   // ============================================================
   // 9. Перевірка положення відносно контрольних точок
   // ============================================================

   // TRUE  - координата знаходиться між контрольними точками.
   // FALSE - координата знаходиться поза ними,
   //         тому використовується лінійна екстраполяція.
   //
   // Вихід за межі контрольних точок НЕ є причиною
   // для заборони розрахунку preset.

   #InConfiguredRange :=
   (#Position_mm >= #PositionMinimum_mm)
   AND
   (#Position_mm <= #PositionMaximum_mm);

   IF NOT #InConfiguredRange THEN

       // Bit 4:
       // Цільова координата знаходиться поза діапазоном
       // двох контрольних точок.
       //
       // Це інформаційний/діагностичний біт.
       // Розрахунок продовжується методом екстраполяції.
       #Status := #Status OR W#16#0010;

   END_IF;


   // ============================================================
   // 10. Перетворення координати у raw
   // ============================================================

   #PositionDelta_mm :=
   #Position_mm
   - #PositionPoint1_mm;


   // Зворотна формула до FC_EncoderScale:
   //
   // Raw = RawPoint1
   //     + (Position - PositionPoint1)
   //       * RawSpan / PositionSpan

   #CalculatedRaw :=
   DINT_TO_LREAL(#RawPoint1)
   +
   (
   #PositionDelta_mm
   * #RawSpan
   / #PositionSpan_mm
   );

   #CalculationValid := TRUE;


   // ============================================================
   // 11. Перевірка фізично допустимого raw-діапазону
   // ============================================================

   // Саме ця перевірка є остаточним обмеженням
   // для можливості виконання hardware preset.

   #InRawRange :=
   (#CalculatedRaw >= DINT_TO_LREAL(#RawMinimum))
   AND
   (#CalculatedRaw <= DINT_TO_LREAL(#RawMaximum));

   IF NOT #InRawRange THEN

       // Bit 5:
       // Розраховане raw знаходиться поза
       // допустимим діапазоном енкодера.
       #Status := #Status OR W#16#0020;

       RETURN;

   END_IF;


   // ============================================================
   // 12. Перетворення розрахованого raw у DINT
   // ============================================================

   // Перетворення виконується тільки після перевірки
   // RawMinimum ... RawMaximum.
   //
   // Оскільки RawMinimum та RawMaximum мають тип DINT,
   // після успішної перевірки значення безпечно
   // перетворювати у DINT.

   #RawPosition :=
   LREAL_TO_DINT(#CalculatedRaw);


   // ============================================================
   // 13. Формування фінальної валідності
   // ============================================================

   // InConfiguredRange тут навмисно НЕ використовується.
   //
   // Координата може знаходитися поза двома контрольними
   // точками масштабування. У такому випадку використовується
   // лінійна екстраполяція.
   //
   // Для дозволу preset необхідно:
   // - коректна конфігурація;
   // - виконаний розрахунок;
   // - розраховане raw знаходиться у допустимих межах.

   #RawPositionValid :=
   #ConfigurationValid
   AND
   #CalculationValid
   AND
   #InRawRange;

   IF #RawPositionValid THEN

       // Bit 7:
       // Raw-значення валідне та може використовуватись
       // для hardware preset енкодера.
       #Status := #Status OR W#16#0080;

   END_IF;
END_FUNCTION

// folder: 700_Calibration/Crane

FUNCTION_BLOCK "FB_CraneCalibration"   // FB703, SCL
{ S7_Optimized_Access := 'TRUE' }
VERSION : 0.1
   VAR_INPUT
      ix_Start : Bool := FALSE;   // Запуск процедури калібровки моста
      ix_Reset : Bool := FALSE;   // Скидання сіквенсера поточної процедури калібровки (без зміни статусу)
      ix_Abort : Bool := FALSE;   // Ручне переривання процедури
      ix_ForceCalibrated : Bool := FALSE;   // Примусове встановлення статусу калібровки для ПНР
      ix_HoistCalibrated : Bool := FALSE;   // Механізм підйому відкалібрований
      ix_TrolleyCalibrated : Bool := FALSE;   // Механізм візка відкалібрований
      il_HoistPosition_mm : LReal := 0.0;   // Поточна координата механізму підйому, мм
      il_HoistPositionMin_mm : LReal := 23750.0;   // Нижня межа допустимого положення підйому для калібровки моста
      il_HoistPositionMax_mm : LReal := 23900.0;   // Верхня межа допустимого положення підйому для калібровки моста
      ix_Reference4K1 : Bool := FALSE;   // Реперний сигнал 4K1 — дозвіл номінальної швидкості при русі вліво
      ix_BtnRight : Bool := FALSE;   // Команда руху моста вправо
      ix_BtnLeft : Bool := FALSE;   // Команда руху моста вліво
      ix_Drive1Fault : Bool := FALSE;   // Аварія частотного перетворювача 4UZ1
      ix_Drive2Fault : Bool := FALSE;   // Аварія частотного перетворювача 4UZ2
      ir_Drive1Velocity_rpm : Real := 0.0;   // Фактична швидкість привода 4UZ1, об/хв
      ir_Drive2Velocity_rpm : Real := 0.0;   // Фактична швидкість привода 4UZ2, об/хв
      ix_Encoder1Ready : Bool := FALSE;   // Енкодер 4BR1 готовий
      ix_Encoder2Ready : Bool := FALSE;   // Енкодер 4BR2 готовий
      ix_Encoder1Fault : Bool := FALSE;   // Помилка енкодера 4BR1
      ix_Encoder2Fault : Bool := FALSE;   // Помилка енкодера 4BR2
      ix_Preset1Busy : Bool := FALSE;   // Виконується preset енкодера 4BR1
      ix_Preset1Done : Bool := FALSE;   // Preset енкодера 4BR1 успішно завершено
      ix_Preset1Error : Bool := FALSE;   // Помилка preset енкодера 4BR1
      iw_Preset1Status : Word := W#16#0000;   // Статус виконання preset енкодера 4BR1
      ix_Preset2Busy : Bool := FALSE;   // Виконується preset енкодера 4BR2
      ix_Preset2Done : Bool := FALSE;   // Preset енкодера 4BR2 успішно завершено
      ix_Preset2Error : Bool := FALSE;   // Помилка preset енкодера 4BR2
      iw_Preset2Status : Word := W#16#0000;   // Статус виконання preset енкодера 4BR2
      id_PresetValueRaw1 : DInt := DINT#11061828;   // Розраховане raw-значення для preset енкодера 4BR1.
      id_PresetValueRaw2 : DInt := DINT#11061828;   // Розраховане raw-значення для preset енкодера 4BR2.
      it_TimeoutA : Time := T#1m;   // Максимальний час очікування першої команди руху
      it_TimeoutB : Time := T#5m;   // Максимальний час виконання реперної процедури
      ir_StandstillSpeed_rpm : Real := 5.0;   // Максимальна швидкість привода для визначення стану standstill
      it_StandstillConfirm : Time := T#500ms;   // Час підтвердження повної зупинки обох приводів
      id_ActualPositionRaw1 : DInt := 0;   // Поточне raw-положення енкодера 4BR1
      id_ActualPositionRaw2 : DInt := 0;   // Поточне raw-положення енкодера 4BR2
      il_Scale1_mm_per_count : LReal := 0.0;   // Масштаб 4BR1, мм/count
      il_Scale2_mm_per_count : LReal := 0.0;   // Масштаб 4BR2, мм/count
      ix_PositionScale1Valid : Bool := FALSE;   // Валідність масштабування 4BR1
      ix_PositionScale2Valid : Bool := FALSE;   // Валідність масштабування 4BR2
   END_VAR
   VAR_OUTPUT
      qx_Active : Bool := FALSE;   // Процедура калібровки моста активна
      qx_Calibrated : Bool := FALSE;   // Механізм моста відкалібрований
      qx_Aborted : Bool := FALSE;   // Процедуру калібровки перервано
      qx_Fault : Bool := FALSE;   // Помилка процедури калібровки
      qx_PrerequisitesNotOK : Bool := FALSE;   // Не виконані попередні умови для калібровки моста
      qu_CurrentStep : UInt := UINT#0;   // Поточний крок сіквенсера калібровки
      qd_CompletedSteps : DWord := DWORD#0;   // Бітова маска завершених кроків калібровки
      qt_StepElapsed : Time := T#0ms;   // Час перебування на поточному кроці
      qt_ActiveTimerElapsed : Time := T#0ms;   // Поточний час активного контрольного таймера
      qt_ActiveTimerPreset : Time := T#0ms;   // Уставка активного контрольного таймера
      qt_ActiveTimerRemaining : Time := T#0ms;   // Залишок часу активного контрольного таймера
      qx_BlockRight : Bool := FALSE;   // Заборона руху моста вправо від сіквенсера калібровки
      qx_BlockLeft : Bool := FALSE;   // Заборона руху моста вліво від сіквенсера калібровки
      qx_QuickStop : Bool := FALSE;   // Запит Quick Stop для обох приводів моста
      qx_DriveStandstill : Bool := FALSE;   // Підтверджена повна зупинка обох приводів
      qx_PresetServiceEnable : Bool := FALSE;   // Загальний дозвіл preset для 4BR1 та 4BR2
      qx_PresetPermit : Bool := FALSE;   // Загальний дозвіл виконання preset для 4BR1 та 4BR2
      qx_PresetStart : Bool := FALSE;   // Загальний одноцикловий запуск preset для 4BR1 та 4BR2
      qd_PresetValueRaw1 : DInt := DINT#0;   // Значення preset, передане енкодеру 4BR1
      qd_PresetValueRaw2 : DInt := DINT#0;   // Значення preset, передане енкодеру 4BR2
      qw_Preset1Status : Word := W#16#0000;   // Поточний статус preset енкодера 4BR1
      qw_Preset2Status : Word := W#16#0000;   // Поточний статус preset енкодера 4BR2
      qw_Status : Word := W#16#0000;   // Загальне діагностичне слово стану блока калібровки
      ql_TravelAfterReference1_mm : LReal := 0.0;   // Шлях, пройдений після повторного проходження 4K1 до повної зупинки (4BR1), мм.
      ql_TravelAfterReference2_mm : LReal := 0.0;   // Шлях, пройдений після повторного проходження 4K1 до повної зупинки (4BR2), мм.
   END_VAR
   VAR
      stat_Step : UInt := UINT#0;   // Поточний внутрішній крок сіквенсера
      stat_PrevStep : UInt := UINT#0;   // Попередній крок для визначення зміни кроку
   END_VAR
   VAR RETAIN
      stat_Calibrated : Bool := FALSE;   // Запам'ятований результат успішної калібровки моста
   END_VAR
   VAR
      stat_MotionStarted : Bool := FALSE;   // Ознака, що під час процедури вже була команда руху
      stat_CompletedSteps : DWord := DWORD#0;   // Внутрішня бітова маска завершених кроків
      stat_StartOld : Bool := FALSE;   // Попередній стан команди Start
      stat_ResetOld : Bool := FALSE;   // Попередній стан команди Reset
      stat_AbortOld : Bool := FALSE;   // Попередній стан команди Abort
      stat_ReferenceOld : Bool := FALSE;   // Попередній стан реперного сигналу 4K1
      tmr_TimeoutA : TON_TIME;   // Таймер очікування першої команди руху
      tmr_TimeoutB : TON_TIME;   // Таймер максимальної тривалості реперної процедури
      tmr_Standstill : TON_TIME;   // Таймер підтвердження повної зупинки обох ПЧ
      tmr_StepElapsed : TON_TIME;   // Таймер часу перебування на поточному кроці
      stat_RawAtReference1 : DInt := 0;   // Raw-положення енкодера 4BR1 в момент повторного спадного фронту 4K1.
      stat_RawAtReference2 : DInt := 0;   // Raw-положення енкодера 4BR2 в момент повторного спадного фронту 4K1.
      stat_RawAtReference1Valid : Bool := FALSE;   // TRUE - raw-положення 4BR1 в точці 4K1 успішно зафіксовано.
      stat_RawAtReference2Valid : Bool := FALSE;   // TRUE - raw-положення 4BR2 в точці 4K1 успішно зафіксовано.
      stat_TravelAfterReference1_mm : LReal := 0.0;   // Розрахований шлях 4BR1 від 4K1 до повної зупинки.
      stat_TravelAfterReference2_mm : LReal := 0.0;   // Розрахований шлях 4BR2 від 4K1 до повної зупинки.
   END_VAR
   VAR_TEMP
      StartEdge : Bool;   // Передній фронт команди запуску калібровки
      ResetEdge : Bool;   // Передній фронт команди Reset
      AbortEdge : Bool;   // Передній фронт команди Abort
      ReferenceFalling : Bool;   // Спадний фронт 4K1, тобто проходження реперної точки при русі вліво
      StepChanged : Bool;   // Ознака зміни поточного кроку сіквенсера
      StandstillCondition : Bool;   // Обидва приводи мають швидкість нижче порога standstill
      HoistPositionOK : Bool;   // Підйом калібрований та знаходиться в допустимій зоні
      PrerequisitesOK : Bool;   // Виконані всі попередні умови для калібровки моста
   END_VAR
BEGIN
   // ============================================================
   // 1. Формування фронтів
   // ============================================================

   #StartEdge :=
   #ix_Start
   AND NOT #stat_StartOld;

   #ResetEdge :=
   #ix_Reset
   AND NOT #stat_ResetOld;

   #AbortEdge :=
   #ix_Abort
   AND NOT #stat_AbortOld;

   // 4K1: проходження репера при русі вліво.
   // Сигнал змінюється TRUE -> FALSE.
   #ReferenceFalling :=
   #stat_ReferenceOld
   AND NOT #ix_Reference4K1;


   // ============================================================
   // 2. Початкові умови калібровки моста
   // ============================================================

   #HoistPositionOK :=
   #ix_HoistCalibrated
   AND (#il_HoistPosition_mm >= #il_HoistPositionMin_mm)
   AND (#il_HoistPosition_mm <= #il_HoistPositionMax_mm);

   #PrerequisitesOK :=
   #HoistPositionOK
   AND #ix_TrolleyCalibrated;

   #qx_PrerequisitesNotOK :=
   NOT #PrerequisitesOK;


   // ============================================================
   // 3. Reset
   // ============================================================

   IF #ResetEdge THEN

       #stat_Step := UINT#0;
       #stat_PrevStep := UINT#0;

       #stat_MotionStarted := FALSE;
       #stat_CompletedSteps := DWORD#0;

       #stat_RawAtReference1 := DINT#0;
       #stat_RawAtReference2 := DINT#0;

       #stat_RawAtReference1Valid := FALSE;
       #stat_RawAtReference2Valid := FALSE;

       #stat_TravelAfterReference1_mm := 0.0;
       #stat_TravelAfterReference2_mm := 0.0;


   END_IF;


   // ============================================================
   // 4. Timeout A
   // ============================================================

   #tmr_TimeoutA(
                 IN :=
                 (#stat_Step = UINT#5)
                 OR (#stat_Step = UINT#20)
                 OR (#stat_Step = UINT#50)
                 OR (#stat_Step = UINT#70),
                 PT := #it_TimeoutA
   );


   // ============================================================
   // 5. Timeout B
   // ============================================================

   #tmr_TimeoutB(
                 IN :=
                 (#stat_Step = UINT#30)
                 OR (#stat_Step = UINT#80),
                 PT := #it_TimeoutB
   );


   // ============================================================
   // 6. Контроль повної зупинки обох приводів
   // ============================================================

   #StandstillCondition :=
   (ABS(#ir_Drive1Velocity_rpm) <= #ir_StandstillSpeed_rpm)
   AND
   (ABS(#ir_Drive2Velocity_rpm) <= #ir_StandstillSpeed_rpm);

   #tmr_Standstill(
                   IN :=
                   (#stat_Step >= UINT#100)
                   AND (#stat_Step <= UINT#120)
                   AND #StandstillCondition,
                   PT := #it_StandstillConfirm
   );

   #qx_DriveStandstill :=
   #tmr_Standstill.Q;


   // ============================================================
   // 7. Таймер поточного кроку
   // ============================================================

   #StepChanged :=
   #stat_Step <> #stat_PrevStep;

   #tmr_StepElapsed(
                    IN :=
                    (#stat_Step > UINT#0)
                    AND (#stat_Step < UINT#130)
                    AND NOT #StepChanged,
                    PT := T#24d
   );

   #qt_StepElapsed :=
   #tmr_StepElapsed.ET;

   IF #StepChanged THEN
       #stat_PrevStep := #stat_Step;
   END_IF;


   // ============================================================
   // 8. Виходи за замовчуванням
   // ============================================================

   #qx_Active := FALSE;
   #qx_Aborted := FALSE;
   #qx_Fault := FALSE;

   #qx_BlockRight := TRUE;
   #qx_BlockLeft := TRUE;

   #qx_QuickStop := FALSE;

   #qx_PresetServiceEnable := FALSE;
   #qx_PresetPermit := FALSE;
   #qx_PresetStart := FALSE;

   #qd_PresetValueRaw1 :=
   #id_PresetValueRaw1;

   #qd_PresetValueRaw2 :=
   #id_PresetValueRaw2;

   #qw_Preset1Status :=
   #iw_Preset1Status;

   #qw_Preset2Status :=
   #iw_Preset2Status;


   // ============================================================
   // 9. Загальні умови аварійного завершення
   //
   // Працюють тільки під час активної процедури.
   // STEP 130 після успішної калібровки не переводиться в 910.
   // ============================================================

   IF (#stat_Step > UINT#0)
       AND (#stat_Step < UINT#130)
   THEN

       IF #AbortEdge THEN

           #stat_Step := UINT#900;

       ELSIF #ix_Drive1Fault
           OR #ix_Drive2Fault
           OR #ix_Encoder1Fault
           OR #ix_Encoder2Fault
       THEN

           #stat_Step := UINT#910;

           // Підйом і візок повинні залишатися
           // у допустимому стані під час процедури.
       ELSIF NOT #PrerequisitesOK THEN

           #stat_Step := UINT#910;

       ELSIF (#stat_Step < UINT#110)
           AND (
           NOT #ix_Encoder1Ready
           OR NOT #ix_Encoder2Ready
           )
       THEN

           #stat_Step := UINT#910;

       ELSIF #tmr_TimeoutA.Q THEN

           #stat_Step := UINT#910;

       ELSIF #tmr_TimeoutB.Q THEN

           #stat_Step := UINT#910;

       END_IF;

   END_IF;


   // ============================================================
   // 10. Основний сіквенсер
   // ============================================================

   CASE #stat_Step OF


           // --------------------------------------------------------
           // STEP 0
           // Калібровка неактивна
           // --------------------------------------------------------
       UINT#0:

           #qx_BlockRight := FALSE;
           #qx_BlockLeft := FALSE;

           IF #StartEdge THEN

               #stat_Calibrated := FALSE;
               #stat_MotionStarted := FALSE;
               #stat_CompletedSteps := DWORD#0;

               #stat_RawAtReference1 := DINT#0;
               #stat_RawAtReference2 := DINT#0;

               #stat_RawAtReference1Valid := FALSE;
               #stat_RawAtReference2Valid := FALSE;

               #stat_TravelAfterReference1_mm := 0.0;
               #stat_TravelAfterReference2_mm := 0.0;

               IF #PrerequisitesOK THEN

                   // Нормальний старт перед репером 4K1.
                   IF #ix_Reference4K1 THEN

                       #stat_Step := UINT#10;

                       // Якщо механізм вже знаходиться на / за 4K1,
                       // спочатку необхідно відійти вправо.
                   ELSE

                       #stat_Step := UINT#5;

                   END_IF;

               ELSE

                   #stat_Step := UINT#910;

               END_IF;

           END_IF;


           // --------------------------------------------------------
           // STEP 5
           // Попередній відхід вправо від 4K1
           // --------------------------------------------------------
       UINT#5:

           #qx_Active := TRUE;

           // До репера вліво рух заборонений.
           // Дозволений тільки відхід вправо.
           #qx_BlockRight := FALSE;
           #qx_BlockLeft := TRUE;

           IF #ix_BtnRight THEN
               #stat_MotionStarted := TRUE;
           END_IF;

           // Після звільнення 4K1 та відпускання кнопки
           // запускаємо штатну процедуру.
           IF #ix_Reference4K1
               AND NOT #ix_BtnRight
           THEN

               #stat_Step := UINT#10;

           END_IF;


           // --------------------------------------------------------
           // STEP 10
           // Перевірка початкових умов
           // --------------------------------------------------------
       UINT#10:

           #qx_Active := TRUE;

           #qx_BlockRight := TRUE;
           #qx_BlockLeft := TRUE;

           IF NOT #ix_BtnRight
               AND NOT #ix_BtnLeft
           THEN

               #stat_CompletedSteps.%X0 := TRUE;
               #stat_Step := UINT#20;

           END_IF;


           // --------------------------------------------------------
           // STEP 20
           // Очікування першої команди "Вліво"
           // --------------------------------------------------------
       UINT#20:

           #qx_Active := TRUE;

           #qx_BlockRight := TRUE;
           #qx_BlockLeft := FALSE;

           IF #ix_BtnLeft THEN

               #stat_MotionStarted := TRUE;
               #stat_CompletedSteps.%X1 := TRUE;

               #stat_Step := UINT#30;

           END_IF;


           // --------------------------------------------------------
           // STEP 30
           // Перший рух вліво до 4K1
           // --------------------------------------------------------
       UINT#30:

           #qx_Active := TRUE;

           #qx_BlockRight := TRUE;
           #qx_BlockLeft := FALSE;

           IF #ReferenceFalling THEN

               #stat_CompletedSteps.%X2 := TRUE;
               #stat_Step := UINT#40;

           END_IF;


           // --------------------------------------------------------
           // STEP 40
           // Перше проходження 4K1
           // Очікування відпускання кнопки "Вліво"
           // --------------------------------------------------------
       UINT#40:

           #qx_Active := TRUE;

           #qx_BlockRight := TRUE;
           #qx_BlockLeft := TRUE;

           IF NOT #ix_BtnLeft THEN

               #stat_CompletedSteps.%X3 := TRUE;
               #stat_Step := UINT#50;

           END_IF;


           // --------------------------------------------------------
           // STEP 50
           // Відхід вправо від репера
           // --------------------------------------------------------
       UINT#50:

           #qx_Active := TRUE;

           #qx_BlockRight := FALSE;
           #qx_BlockLeft := TRUE;

           IF #ix_BtnRight THEN
               #stat_MotionStarted := TRUE;
           END_IF;

           IF #ix_Reference4K1
               AND NOT #ix_BtnRight
           THEN

               #stat_CompletedSteps.%X4 := TRUE;
               #stat_Step := UINT#60;

           END_IF;


           // --------------------------------------------------------
           // STEP 60
           // Репер звільнений
           // --------------------------------------------------------
       UINT#60:

           #qx_Active := TRUE;

           #qx_BlockRight := TRUE;
           #qx_BlockLeft := TRUE;

           #stat_CompletedSteps.%X5 := TRUE;
           #stat_Step := UINT#70;


           // --------------------------------------------------------
           // STEP 70
           // Очікування повторної команди "Вліво"
           // --------------------------------------------------------
       UINT#70:

           #qx_Active := TRUE;

           #qx_BlockRight := TRUE;
           #qx_BlockLeft := FALSE;

           IF #ix_BtnLeft THEN

               #stat_CompletedSteps.%X6 := TRUE;
               #stat_Step := UINT#80;

           END_IF;


           // --------------------------------------------------------
           // STEP 80
           // Повторний точний підхід вліво до 4K1
           // --------------------------------------------------------
       UINT#80:

           #qx_Active := TRUE;

           #qx_BlockRight := TRUE;
           #qx_BlockLeft := FALSE;

           IF #ReferenceFalling THEN

               // Обидва канали масштабування повинні бути валідні.
               IF #ix_PositionScale1Valid
                   AND #ix_PositionScale2Valid
               THEN

                   // Одночасно запам'ятовуємо raw-положення
                   // обох енкодерів у момент проходження 4K1.
                   #stat_RawAtReference1 :=
                   #id_ActualPositionRaw1;

                   #stat_RawAtReference2 :=
                   #id_ActualPositionRaw2;

                   #stat_RawAtReference1Valid := TRUE;
                   #stat_RawAtReference2Valid := TRUE;

                   #stat_CompletedSteps.%X7 := TRUE;
                   #stat_Step := UINT#90;

               ELSE

                   #stat_RawAtReference1Valid := FALSE;
                   #stat_RawAtReference2Valid := FALSE;

                   #stat_Step := UINT#910;

               END_IF;

           END_IF;



           // --------------------------------------------------------
           // STEP 90
           // Quick Stop обох приводів
           // --------------------------------------------------------
       UINT#90:

           #qx_Active := TRUE;

           #qx_BlockRight := TRUE;
           #qx_BlockLeft := TRUE;
           #qx_QuickStop := TRUE;

           #stat_CompletedSteps.%X8 := TRUE;

           #stat_Step := UINT#100;


           // --------------------------------------------------------
           // STEP 100
           // Очікування повної зупинки обох приводів
           // --------------------------------------------------------
       UINT#100:

           #qx_Active := TRUE;

           #qx_BlockRight := TRUE;
           #qx_BlockLeft := TRUE;

           #qx_QuickStop := TRUE;

           IF #qx_DriveStandstill
               AND NOT #ix_BtnRight
               AND NOT #ix_BtnLeft
           THEN

               IF #stat_RawAtReference1Valid
                   AND #stat_RawAtReference2Valid
                   AND #ix_PositionScale1Valid
                   AND #ix_PositionScale2Valid
               THEN

                   // Шлях 4BR1 від проходження 4K1
                   // до підтвердженої повної зупинки.
                   #stat_TravelAfterReference1_mm :=
                   (
                   DINT_TO_LREAL(#id_ActualPositionRaw1)
                   - DINT_TO_LREAL(#stat_RawAtReference1)
                   )
                   * #il_Scale1_mm_per_count;

                   // Шлях 4BR2 від проходження 4K1
                   // до підтвердженої повної зупинки.
                   #stat_TravelAfterReference2_mm :=
                   (
                   DINT_TO_LREAL(#id_ActualPositionRaw2)
                   - DINT_TO_LREAL(#stat_RawAtReference2)
                   )
                   * #il_Scale2_mm_per_count;

                   #stat_CompletedSteps.%X9 := TRUE;
                   #stat_Step := UINT#110;

               ELSE

                   #stat_Step := UINT#910;

               END_IF;

           END_IF;


           // --------------------------------------------------------
           // STEP 110
           // Запуск preset обох енкодерів
           // --------------------------------------------------------
       UINT#110:

           #qx_Active := TRUE;

           #qx_BlockRight := TRUE;
           #qx_BlockLeft := TRUE;

           #qx_PresetServiceEnable := TRUE;

           #qx_PresetPermit :=
           #qx_DriveStandstill
           AND NOT #ix_BtnRight
           AND NOT #ix_BtnLeft
           AND #ix_Encoder1Ready
           AND #ix_Encoder2Ready
           AND NOT #ix_Encoder1Fault
           AND NOT #ix_Encoder2Fault
           AND NOT #ix_Drive1Fault
           AND NOT #ix_Drive2Fault;

           IF #qx_PresetPermit THEN

               // Один імпульс одночасно запускає preset
               // для 4BR1 та 4BR2.
               #qx_PresetStart := TRUE;

               #stat_CompletedSteps.%X10 := TRUE;
               #stat_Step := UINT#120;

           END_IF;


           // --------------------------------------------------------
           // STEP 120
           // Очікування завершення preset обох енкодерів
           // --------------------------------------------------------
       UINT#120:

           #qx_Active := TRUE;

           #qx_BlockRight := TRUE;
           #qx_BlockLeft := TRUE;

           #qx_PresetServiceEnable := TRUE;

           #qx_PresetPermit :=
           #qx_DriveStandstill
           AND NOT #ix_BtnRight
           AND NOT #ix_BtnLeft
           AND NOT #ix_Encoder1Fault
           AND NOT #ix_Encoder2Fault
           AND NOT #ix_Drive1Fault
           AND NOT #ix_Drive2Fault;

           // Обидва preset повинні завершитися успішно.
           IF #ix_Preset1Done
               AND #ix_Preset2Done
           THEN

               #stat_CompletedSteps.%X11 := TRUE;
               #stat_Step := UINT#130;

           ELSIF #ix_Preset1Error
               OR #ix_Preset2Error
           THEN

               #stat_Step := UINT#910;

           END_IF;


           // --------------------------------------------------------
           // STEP 130
           // Калібровка моста успішно завершена
           // --------------------------------------------------------
       UINT#130:

           #qx_BlockRight := FALSE;
           #qx_BlockLeft := FALSE;

           #stat_Calibrated := TRUE;
           #stat_CompletedSteps.%X12 := TRUE;


           // --------------------------------------------------------
           // STEP 900
           // Ручне переривання
           // --------------------------------------------------------
       UINT#900:

           #qx_Aborted := TRUE;

           #qx_BlockRight := TRUE;
           #qx_BlockLeft := TRUE;

           #qx_QuickStop := TRUE;


           // --------------------------------------------------------
           // STEP 910
           // Помилка процедури
           // --------------------------------------------------------
       UINT#910:

           #qx_Fault := TRUE;

           #qx_BlockRight := TRUE;
           #qx_BlockLeft := TRUE;

           #qx_QuickStop := TRUE;


       ELSE

           #stat_Step := UINT#910;

   END_CASE;


   // ============================================================
   // 11. Основні статуси
   // ============================================================

   #qu_CurrentStep :=
   #stat_Step;

   #qd_CompletedSteps :=
   #stat_CompletedSteps;

   #qx_Calibrated :=
   #stat_Calibrated
   OR #ix_ForceCalibrated;

   #ql_TravelAfterReference1_mm :=
   #stat_TravelAfterReference1_mm;

   #ql_TravelAfterReference2_mm :=
   #stat_TravelAfterReference2_mm;

   // ============================================================
   // 12. Активний таймер для HMI
   // ============================================================

   #qt_ActiveTimerElapsed := T#0ms;
   #qt_ActiveTimerPreset := T#0ms;
   #qt_ActiveTimerRemaining := T#0ms;

   // Timeout A
   IF (#stat_Step = UINT#5)
       OR (#stat_Step = UINT#20)
       OR (#stat_Step = UINT#50)
       OR (#stat_Step = UINT#70)
   THEN

       #qt_ActiveTimerElapsed :=
       #tmr_TimeoutA.ET;

       #qt_ActiveTimerPreset :=
       #it_TimeoutA;

       IF #tmr_TimeoutA.ET < #it_TimeoutA THEN

           #qt_ActiveTimerRemaining :=
           #it_TimeoutA - #tmr_TimeoutA.ET;

       END_IF;


       // Timeout B
   ELSIF 
       (#stat_Step = UINT#30)
       OR (#stat_Step = UINT#80)
   THEN

       #qt_ActiveTimerElapsed :=
       #tmr_TimeoutB.ET;

       #qt_ActiveTimerPreset :=
       #it_TimeoutB;

       IF #tmr_TimeoutB.ET < #it_TimeoutB THEN

           #qt_ActiveTimerRemaining :=
           #it_TimeoutB - #tmr_TimeoutB.ET;

       END_IF;


       // Standstill
   ELSIF #stat_Step = UINT#100 THEN

       #qt_ActiveTimerElapsed :=
       #tmr_Standstill.ET;

       #qt_ActiveTimerPreset :=
       #it_StandstillConfirm;

       IF #tmr_Standstill.ET < #it_StandstillConfirm THEN

           #qt_ActiveTimerRemaining :=
           #it_StandstillConfirm - #tmr_Standstill.ET;

       END_IF;

   END_IF;


   // ============================================================
   // 13. Діагностичне слово
   // ============================================================

   #qw_Status := W#16#0000;

   IF #qx_Active THEN
       #qw_Status := #qw_Status OR W#16#0001;
   END_IF;

   IF #qx_Calibrated THEN
       #qw_Status := #qw_Status OR W#16#0002;
   END_IF;

   IF #qx_Aborted THEN
       #qw_Status := #qw_Status OR W#16#0004;
   END_IF;

   IF #qx_Fault THEN
       #qw_Status := #qw_Status OR W#16#0008;
   END_IF;

   IF #qx_DriveStandstill THEN
       #qw_Status := #qw_Status OR W#16#0010;
   END_IF;

   IF #ix_Preset1Busy OR #ix_Preset2Busy THEN
       #qw_Status := #qw_Status OR W#16#0020;
   END_IF;

   IF #ix_Preset1Error OR #ix_Preset2Error THEN
       #qw_Status := #qw_Status OR W#16#0040;
   END_IF;

   IF #qx_PrerequisitesNotOK THEN
       #qw_Status := #qw_Status OR W#16#0080;
   END_IF;

   IF #tmr_TimeoutA.Q THEN
       #qw_Status := #qw_Status OR W#16#0100;
   END_IF;

   IF #tmr_TimeoutB.Q THEN
       #qw_Status := #qw_Status OR W#16#0200;
   END_IF;

   IF #ix_Drive1Fault OR #ix_Drive2Fault THEN
       #qw_Status := #qw_Status OR W#16#0400;
   END_IF;

   IF #ix_Encoder1Fault OR #ix_Encoder2Fault THEN
       #qw_Status := #qw_Status OR W#16#0800;
   END_IF;

   IF NOT #ix_Encoder1Ready
       OR NOT #ix_Encoder2Ready
   THEN
       #qw_Status := #qw_Status OR W#16#1000;
   END_IF;


   // ============================================================
   // 14. Запам'ятовування станів
   // ============================================================

   #stat_StartOld :=
   #ix_Start;

   #stat_ResetOld :=
   #ix_Reset;

   #stat_AbortOld :=
   #ix_Abort;

   #stat_ReferenceOld :=
   #ix_Reference4K1;
END_FUNCTION_BLOCK

FUNCTION_BLOCK "FB_CraneCalibrationDiag"   // FB713, SCL
{ S7_Optimized_Access := 'TRUE' }
VERSION : 0.1
   VAR_INPUT
      ix_Reset : Bool := FALSE;   // Скидання зафіксованих діагностичних помилок
      ix_Encoder1Ready : Bool := FALSE;   // Енкодер 4BR1 готовий
      ix_Encoder1Fault : Bool := FALSE;   // Помилка енкодера 4BR1
      ix_Communication1Fault : Bool := FALSE;   // Помилка зв'язку з енкодером 4BR1
      il_Position1_mm : LReal := 0.0;   // Поточна координата за енкодером 4BR1, мм
      ix_Encoder2Ready : Bool := FALSE;   // Енкодер 4BR2 готовий
      ix_Encoder2Fault : Bool := FALSE;   // Помилка енкодера 4BR2
      ix_Communication2Fault : Bool := FALSE;   // Помилка зв'язку з енкодером 4BR2
      il_Position2_mm : LReal := 0.0;   // Поточна координата за енкодером 4BR2, мм
      ix_MoveCommand : Bool := FALSE;   // Дійсна команда руху моста
      ix_Drive1Fault : Bool := FALSE;   // Аварія привода 4UZ1
      ix_Drive2Fault : Bool := FALSE;   // Аварія привода 4UZ2
      ir_Drive1Velocity_rpm : Real := 0.0;   // Фактична швидкість 4UZ1, об/хв
      ir_Drive2Velocity_rpm : Real := 0.0;   // Фактична швидкість 4UZ2, об/хв
      ix_CalibrationActive : Bool := FALSE;   // Процедура калібровки моста активна
      ix_Calibrated : Bool := FALSE;   // Міст відкалібрований
      ix_ManualDriveActive : Bool := FALSE;   // Ручний привод активний; поки FALSE
      il_NoMoveThreshold_mm : LReal := 5.0;   // Допустима зміна положення без команди
      il_MoveMinDelta_mm : LReal := 1.0;   // Мінімальна зміна координати при русі
      it_MoveUpdateTimeout : Time := T#1s;   // Максимальний час без зміни координати
      ir_StandstillSpeed_rpm : Real := 5.0;   // Поріг повної зупинки приводів
      it_StandstillConfirm : Time := T#500ms;   // Час підтвердження повної зупинки
      il_StartupTolerance_mm : LReal := 5.0;   // Допуск перевірки координати після запуску PLC
      il_MaxEncoderDifference_mm : LReal := 50.0;   // Максимальна допустима розбіжність 4BR1 та 4BR2
   END_VAR
   VAR_OUTPUT
      qx_Encoder1ControlHealthy : Bool := FALSE;   // Енкодер 4BR1 і його зв'язок справні
      qx_Encoder1StartupDataConsistent : Bool := TRUE;   // Дані 4BR1 після старту PLC узгоджені
      qx_Encoder1NoMovementWithoutCommand : Bool := TRUE;   // Для 4BR1 не виявлено руху без команди
      qx_Encoder1NoManualMovementDetected : Bool := TRUE;   // Для 4BR1 не виявлено нештатного переміщення
      qx_Encoder1UpdatesDuringMotion : Bool := TRUE;   // 4BR1 змінює координату під час руху
      qx_Encoder1ReplacementNotDetected : Bool := TRUE;   // Заміна 4BR1 не виявлена; поки завжди норма
      qx_Encoder2ControlHealthy : Bool := FALSE;   // Енкодер 4BR2 і його зв'язок справні
      qx_Encoder2StartupDataConsistent : Bool := TRUE;   // Дані 4BR2 після старту PLC узгоджені
      qx_Encoder2NoMovementWithoutCommand : Bool := TRUE;   // Для 4BR2 не виявлено руху без команди
      qx_Encoder2NoManualMovementDetected : Bool := TRUE;   // Для 4BR2 не виявлено нештатного переміщення
      qx_Encoder2UpdatesDuringMotion : Bool := TRUE;   // 4BR2 змінює координату під час руху
      qx_Encoder2ReplacementNotDetected : Bool := TRUE;   // Заміна 4BR2 не виявлена; поки завжди норма
      qx_EncoderDifferenceOK : Bool := TRUE;   // Розбіжність координат 4BR1/4BR2 у нормі
      qx_DiagnosticsHealthy : Bool := FALSE;   // Загальний результат діагностики моста
      qx_DriveStandstill : Bool := FALSE;   // Підтверджена повна зупинка обох приводів
      ql_EncoderDifference_mm : LReal := 0.0;   // Поточна абсолютна розбіжність 4BR1/4BR2, мм
      ql_Position1DeltaStopped_mm : LReal := 0.0;   // Зміна 4BR1 від точки зупинки
      ql_Position2DeltaStopped_mm : LReal := 0.0;   // Зміна 4BR2 від точки зупинки
      ql_Position1DeltaMotion_mm : LReal := 0.0;   // Зміна 4BR1 для watchdog руху
      ql_Position2DeltaMotion_mm : LReal := 0.0;   // Зміна 4BR2 для watchdog руху
   END_VAR
   VAR RETAIN
      stat_SavedPosition1_mm : LReal := 0.0;   // Збережена до перезапуску позиція 4BR1
      stat_SavedPosition1Valid : Bool := FALSE;   // Збережена позиція 4BR1 валідна
      stat_SavedPosition2_mm : LReal := 0.0;   // Збережена до перезапуску позиція 4BR2
      stat_SavedPosition2Valid : Bool := FALSE;   // Збережена позиція 4BR2 валідна
   END_VAR
   VAR
      stat_StartupChecked : Bool := FALSE;   // Стартова перевірка виконана
      stat_StopReference1_mm : LReal := 0.0;   // Базова позиція 4BR1 після зупинки
      stat_StopReference1Valid : Bool := FALSE;   // Базова позиція 4BR1 валідна
      stat_StopReference2_mm : LReal := 0.0;   // Базова позиція 4BR2 після зупинки
      stat_StopReference2Valid : Bool := FALSE;   // Базова позиція 4BR2 валідна
      stat_MoveReference1_mm : LReal := 0.0;   // База watchdog 4BR1
      stat_MoveReference2_mm : LReal := 0.0;   // База watchdog 4BR2
      stat_MoveMonitor1Active : Bool := FALSE;   // Watchdog 4BR1 активний
      stat_MoveMonitor2Active : Bool := FALSE;   // Watchdog 4BR2 активний
      stat_WasMoving : Bool := FALSE;   // Міст до цього рухався
      stat_StartupMismatch1Fault : Bool := FALSE;   // Стартова невідповідність 4BR1
      stat_StartupMismatch2Fault : Bool := FALSE;   // Стартова невідповідність 4BR2
      stat_MoveWithoutCommand1Fault : Bool := FALSE;   // Зміна 4BR1 без команди
      stat_MoveWithoutCommand2Fault : Bool := FALSE;   // Зміна 4BR2 без команди
      stat_NoUpdateDuringMotion1Fault : Bool := FALSE;   // 4BR1 не оновлюється при русі
      stat_NoUpdateDuringMotion2Fault : Bool := FALSE;   // 4BR2 не оновлюється при русі
      stat_EncoderDifferenceFault : Bool := FALSE;   // Розбіжність енкодерів перевищила допустиму
      stat_CalibratedOld : Bool := FALSE;   // Попередній стан Calibrated
      tmr_Standstill : TON_TIME;   // Підтвердження повної зупинки
      tmr_MoveUpdate1 : TON_TIME;   // Watchdog 4BR1
      tmr_MoveUpdate2 : TON_TIME;   // Watchdog 4BR2
   END_VAR
   VAR_TEMP
      Encoder1Healthy : Bool;   // Поточна справність 4BR1
      Encoder2Healthy : Bool;   // Поточна справність 4BR2
      StandstillCondition : Bool;   // Обидва ПЧ мають низьку швидкість
      CalibratedRising : Bool;   // Передній фронт Calibrated
      MoveDelta1Reached : Bool;   // 4BR1 змінився на задану величину
      MoveDelta2Reached : Bool;   // 4BR2 змінився на задану величину
      MoveWatchdog1Enable : Bool;   // Дозвіл watchdog 4BR1
      MoveWatchdog2Enable : Bool;   // Дозвіл watchdog 4BR2
   END_VAR
BEGIN
   // ============================================================
   // 1. Справність енкодерів
   // ============================================================

   #Encoder1Healthy :=
   #ix_Encoder1Ready
   AND NOT #ix_Encoder1Fault
   AND NOT #ix_Communication1Fault;

   #Encoder2Healthy :=
   #ix_Encoder2Ready
   AND NOT #ix_Encoder2Fault
   AND NOT #ix_Communication2Fault;

   #qx_Encoder1ControlHealthy :=
   #Encoder1Healthy;

   #qx_Encoder2ControlHealthy :=
   #Encoder2Healthy;


   // ============================================================
   // 2. Визначення повної зупинки обох приводів
   // ============================================================

   #StandstillCondition :=
   (ABS(#ir_Drive1Velocity_rpm) <= #ir_StandstillSpeed_rpm)
   AND
   (ABS(#ir_Drive2Velocity_rpm) <= #ir_StandstillSpeed_rpm);

   #tmr_Standstill(
                   IN :=
                   #StandstillCondition
                   AND NOT #ix_MoveCommand,
                   PT := #it_StandstillConfirm
   );

   #qx_DriveStandstill :=
   #tmr_Standstill.Q;


   // ============================================================
   // 3. Фронт статусу "Калібровано"
   // ============================================================

   #CalibratedRising :=
   #ix_Calibrated
   AND NOT #stat_CalibratedOld;


   // ============================================================
   // 4. Reset діагностики
   // ============================================================

   IF #ix_Reset THEN

       #stat_StartupMismatch1Fault := FALSE;
       #stat_StartupMismatch2Fault := FALSE;

       #stat_MoveWithoutCommand1Fault := FALSE;
       #stat_MoveWithoutCommand2Fault := FALSE;

       #stat_NoUpdateDuringMotion1Fault := FALSE;
       #stat_NoUpdateDuringMotion2Fault := FALSE;

       #stat_EncoderDifferenceFault := FALSE;

       #stat_StopReference1Valid := FALSE;
       #stat_StopReference2Valid := FALSE;

       #stat_MoveMonitor1Active := FALSE;
       #stat_MoveMonitor2Active := FALSE;

   END_IF;


   // ============================================================
   // 5. Перевірка позицій після запуску PLC
   // ============================================================

   IF NOT #stat_StartupChecked
       AND #Encoder1Healthy
       AND #Encoder2Healthy
   THEN

       // 4BR1
       IF #stat_SavedPosition1Valid THEN

           IF ABS(#il_Position1_mm - #stat_SavedPosition1_mm)
               > #il_StartupTolerance_mm
           THEN
               #stat_StartupMismatch1Fault := TRUE;
           END_IF;

       ELSE

           #stat_SavedPosition1_mm :=
           #il_Position1_mm;

           #stat_SavedPosition1Valid := TRUE;

       END_IF;


       // 4BR2
       IF #stat_SavedPosition2Valid THEN

           IF ABS(#il_Position2_mm - #stat_SavedPosition2_mm)
               > #il_StartupTolerance_mm
           THEN
               #stat_StartupMismatch2Fault := TRUE;
           END_IF;

       ELSE

           #stat_SavedPosition2_mm :=
           #il_Position2_mm;

           #stat_SavedPosition2Valid := TRUE;

       END_IF;


       #stat_StartupChecked := TRUE;

       #stat_StopReference1_mm :=
       #il_Position1_mm;

       #stat_StopReference1Valid := TRUE;

       #stat_StopReference2_mm :=
       #il_Position2_mm;

       #stat_StopReference2Valid := TRUE;

   END_IF;


   // ============================================================
   // 6. Після успішної калібровки
   // ============================================================

   IF #CalibratedRising
       AND #Encoder1Healthy
       AND #Encoder2Healthy
   THEN

       #stat_StopReference1_mm :=
       #il_Position1_mm;

       #stat_StopReference1Valid := TRUE;

       #stat_StopReference2_mm :=
       #il_Position2_mm;

       #stat_StopReference2Valid := TRUE;


       #stat_SavedPosition1_mm :=
       #il_Position1_mm;

       #stat_SavedPosition1Valid := TRUE;

       #stat_SavedPosition2_mm :=
       #il_Position2_mm;

       #stat_SavedPosition2Valid := TRUE;


       #stat_StartupMismatch1Fault := FALSE;
       #stat_StartupMismatch2Fault := FALSE;

       #stat_MoveWithoutCommand1Fault := FALSE;
       #stat_MoveWithoutCommand2Fault := FALSE;

       #stat_NoUpdateDuringMotion1Fault := FALSE;
       #stat_NoUpdateDuringMotion2Fault := FALSE;

       #stat_EncoderDifferenceFault := FALSE;

   END_IF;


   // ============================================================
   // 7. Запам'ятовування факту руху
   // ============================================================

   IF #ix_MoveCommand THEN
       #stat_WasMoving := TRUE;
   END_IF;


   // ============================================================
   // 8. Формування нових баз після завершення руху
   // ============================================================

   IF #qx_DriveStandstill
       AND #stat_WasMoving
       AND #Encoder1Healthy
       AND #Encoder2Healthy
       AND NOT #ix_CalibrationActive
   THEN

       #stat_StopReference1_mm :=
       #il_Position1_mm;

       #stat_StopReference1Valid := TRUE;

       #stat_StopReference2_mm :=
       #il_Position2_mm;

       #stat_StopReference2Valid := TRUE;


       #stat_SavedPosition1_mm :=
       #il_Position1_mm;

       #stat_SavedPosition1Valid := TRUE;

       #stat_SavedPosition2_mm :=
       #il_Position2_mm;

       #stat_SavedPosition2Valid := TRUE;

       #stat_WasMoving := FALSE;

   END_IF;


   // ============================================================
   // 9. Контроль зміни положення без команди
   // ============================================================

   #ql_Position1DeltaStopped_mm := 0.0;
   #ql_Position2DeltaStopped_mm := 0.0;

   IF #qx_DriveStandstill
       AND NOT #ix_MoveCommand
       AND NOT #ix_ManualDriveActive
       AND NOT #ix_CalibrationActive
   THEN

       // 4BR1
       IF #Encoder1Healthy
           AND #stat_StopReference1Valid
       THEN

           #ql_Position1DeltaStopped_mm :=
           ABS(#il_Position1_mm - #stat_StopReference1_mm);

           IF #ql_Position1DeltaStopped_mm
               > #il_NoMoveThreshold_mm
           THEN

               #stat_MoveWithoutCommand1Fault := TRUE;

           END_IF;

       END_IF;


       // 4BR2
       IF #Encoder2Healthy
           AND #stat_StopReference2Valid
       THEN

           #ql_Position2DeltaStopped_mm :=
           ABS(#il_Position2_mm - #stat_StopReference2_mm);

           IF #ql_Position2DeltaStopped_mm
               > #il_NoMoveThreshold_mm
           THEN

               #stat_MoveWithoutCommand2Fault := TRUE;

           END_IF;

       END_IF;

   END_IF;


   // ============================================================
   // 10. Watchdog оновлення 4BR1 під час руху
   // ============================================================

   IF #ix_MoveCommand
       AND NOT #ix_Drive1Fault
       AND #Encoder1Healthy
   THEN

       IF NOT #stat_MoveMonitor1Active THEN

           #stat_MoveReference1_mm :=
           #il_Position1_mm;

           #stat_MoveMonitor1Active := TRUE;

       END_IF;

       #ql_Position1DeltaMotion_mm :=
       ABS(#il_Position1_mm - #stat_MoveReference1_mm);

       #MoveDelta1Reached :=
       #ql_Position1DeltaMotion_mm >= #il_MoveMinDelta_mm;

       IF #MoveDelta1Reached THEN

           #stat_MoveReference1_mm :=
           #il_Position1_mm;

       END_IF;

   ELSE

       #stat_MoveMonitor1Active := FALSE;
       #ql_Position1DeltaMotion_mm := 0.0;
       #MoveDelta1Reached := FALSE;

   END_IF;

   #MoveWatchdog1Enable :=
   #stat_MoveMonitor1Active
   AND NOT #MoveDelta1Reached;

   #tmr_MoveUpdate1(
                    IN := #MoveWatchdog1Enable,
                    PT := #it_MoveUpdateTimeout
   );

   IF #tmr_MoveUpdate1.Q THEN
       #stat_NoUpdateDuringMotion1Fault := TRUE;
   END_IF;


   // ============================================================
   // 11. Watchdog оновлення 4BR2 під час руху
   // ============================================================

   IF #ix_MoveCommand
       AND NOT #ix_Drive2Fault
       AND #Encoder2Healthy
   THEN

       IF NOT #stat_MoveMonitor2Active THEN

           #stat_MoveReference2_mm :=
           #il_Position2_mm;

           #stat_MoveMonitor2Active := TRUE;

       END_IF;

       #ql_Position2DeltaMotion_mm :=
       ABS(#il_Position2_mm - #stat_MoveReference2_mm);

       #MoveDelta2Reached :=
       #ql_Position2DeltaMotion_mm >= #il_MoveMinDelta_mm;

       IF #MoveDelta2Reached THEN

           #stat_MoveReference2_mm :=
           #il_Position2_mm;

       END_IF;

   ELSE

       #stat_MoveMonitor2Active := FALSE;
       #ql_Position2DeltaMotion_mm := 0.0;
       #MoveDelta2Reached := FALSE;

   END_IF;

   #MoveWatchdog2Enable :=
   #stat_MoveMonitor2Active
   AND NOT #MoveDelta2Reached;

   #tmr_MoveUpdate2(
                    IN := #MoveWatchdog2Enable,
                    PT := #it_MoveUpdateTimeout
   );

   IF #tmr_MoveUpdate2.Q THEN
       #stat_NoUpdateDuringMotion2Fault := TRUE;
   END_IF;


   // ============================================================
   // 12. Контроль розбіжності енкодерів моста
   // ============================================================

   #ql_EncoderDifference_mm :=
   ABS(#il_Position1_mm - #il_Position2_mm);

   IF #ix_Calibrated
       AND #Encoder1Healthy
       AND #Encoder2Healthy
       AND (#ql_EncoderDifference_mm > #il_MaxEncoderDifference_mm)
   THEN

       #stat_EncoderDifferenceFault := TRUE;

   END_IF;


   // ============================================================
   // 13. Позитивні діагностичні виходи 4BR1
   // ============================================================

   #qx_Encoder1StartupDataConsistent :=
   NOT #stat_StartupMismatch1Fault;

   #qx_Encoder1NoMovementWithoutCommand :=
   NOT #stat_MoveWithoutCommand1Fault;

   #qx_Encoder1NoManualMovementDetected :=
   NOT #stat_MoveWithoutCommand1Fault;

   #qx_Encoder1UpdatesDuringMotion :=
   NOT #stat_NoUpdateDuringMotion1Fault;

   // Контроль фізичної заміни поки не реалізований.
   #qx_Encoder1ReplacementNotDetected := TRUE;


   // ============================================================
   // 14. Позитивні діагностичні виходи 4BR2
   // ============================================================

   #qx_Encoder2StartupDataConsistent :=
   NOT #stat_StartupMismatch2Fault;

   #qx_Encoder2NoMovementWithoutCommand :=
   NOT #stat_MoveWithoutCommand2Fault;

   #qx_Encoder2NoManualMovementDetected :=
   NOT #stat_MoveWithoutCommand2Fault;

   #qx_Encoder2UpdatesDuringMotion :=
   NOT #stat_NoUpdateDuringMotion2Fault;

   // Контроль фізичної заміни поки не реалізований.
   #qx_Encoder2ReplacementNotDetected := TRUE;


   // ============================================================
   // 15. Розбіжність енкодерів
   // ============================================================

   #qx_EncoderDifferenceOK :=
   NOT #stat_EncoderDifferenceFault;


   // ============================================================
   // 16. Загальний результат діагностики
   // ============================================================

   #qx_DiagnosticsHealthy :=
   #qx_Encoder1ControlHealthy
   AND #qx_Encoder1StartupDataConsistent
   AND #qx_Encoder1NoMovementWithoutCommand
   AND #qx_Encoder1NoManualMovementDetected
   AND #qx_Encoder1UpdatesDuringMotion

   AND #qx_Encoder2ControlHealthy
   AND #qx_Encoder2StartupDataConsistent
   AND #qx_Encoder2NoMovementWithoutCommand
   AND #qx_Encoder2NoManualMovementDetected
   AND #qx_Encoder2UpdatesDuringMotion

   AND #qx_EncoderDifferenceOK;


   // ============================================================
   // 17. Запам'ятовування станів
   // ============================================================

   #stat_CalibratedOld :=
   #ix_Calibrated;
END_FUNCTION_BLOCK

// folder: 700_Calibration/Hoist/Lifting

FUNCTION_BLOCK "FB_HoistCalibration"   // FB701, SCL
{ S7_Optimized_Access := 'TRUE' }
VERSION : 0.1
   VAR_INPUT
      ix_Start : Bool := FALSE;   // Запуск процедури калібровки
      ix_Reset : Bool := FALSE;   // Скидання сіквенсера поточної процедури калібровки (статус не скидається)
      ix_Abort : Bool := FALSE;   // Ручне переривання процедури
      ix_ForceCalibrated : Bool := FALSE;   // Примусове встановлення статусу калібровки для ПНР
      ix_Reference1K1 : Bool := FALSE;   // Сигнал технологічного передзупину 1K1
      ix_BtnUp : Bool := FALSE;   // Команда оператора «Підйом»
      ix_BtnDown : Bool := FALSE;   // Команда оператора «Опускання»
      ix_DriveFault : Bool := FALSE;   // Аварія ПЧ
      ir_DriveVelocity_rpm : Real := 0.0;   // Фактична швидкість ПЧ, об/хв
      ix_EncoderReady : Bool := FALSE;   // Енкодер готовий до роботи
      ix_EncoderFault : Bool := FALSE;   // Активна помилка енкодера
      ix_PresetBusy : Bool := FALSE;   // Процедура preset активна
      ix_PresetDone : Bool := FALSE;   // Імпульс успішного завершення preset
      ix_PresetError : Bool := FALSE;   // Помилка процедури preset
      iw_PresetStatus : Word := W#16#0000;   // Діагностичний код процедури preset
      id_PresetValueRaw : DInt := DINT#130250000;   // Розраховане raw-значення для preset енкодера 1BR.
      it_TimeoutA : Time := T#1m;   // Максимальний час очікування початку руху
      it_TimeoutB : Time := T#5m;   // Максимальний час виконання пошуку реперної точки
      ir_StandstillSpeed_rpm : Real := 5.0;   // Максимальна швидкість для визначення зупинки ПЧ
      it_StandstillConfirm : Time := T#500ms;   // Час підтвердження стану повної зупинки
      id_ActualPositionRaw : DInt := DINT#0;   // Поточне абсолютне raw-положення енкодера 1BR.
      il_Scale_mm_per_count : LReal := 0.0;   // Коефіцієнт перетворення raw-count у мм для енкодера 1BR.
      ix_PositionScaleValid : Bool := FALSE;   // TRUE - масштабування положення енкодера налаштоване коректно.
   END_VAR
   VAR_OUTPUT
      qx_Active : Bool := FALSE;   // Процедура калібровки активна
      qx_Calibrated : Bool := FALSE;   // Механізм має статус «Калібровано»
      qx_Aborted : Bool := FALSE;   // Процедуру калібровки перервано
      qx_Fault : Bool := FALSE;   // Помилка процедури калібровки
      qu_CurrentStep : UInt := UINT#0;   // Поточний номер кроку сіквенсера
      qd_CompletedSteps : DWord := DWORD#0;   // Бітова маска успішно завершених кроків
      qt_StepElapsed : Time := T#0ms;   // Час перебування на поточному кроці
      qt_ActiveTimerElapsed : Time := T#0ms;   // Поточне значення активного таймера
      qt_ActiveTimerPreset : Time := T#0ms;   // Уставка активного таймера
      qt_ActiveTimerRemaining : Time := T#0ms;   // Час до завершення активного таймера
      qx_BlockUp : Bool := FALSE;   // Заборона руху механізму вгору
      qx_BlockDown : Bool := FALSE;   // Заборона руху механізму вниз
      qx_QuickStop : Bool := FALSE;   // Запит Quick Stop / OFF3
      qx_DriveStandstill : Bool := FALSE;   // Підтверджений стан зупинки ПЧ
      qx_PresetServiceEnable : Bool := FALSE;   // Дозвіл сервісної функції preset
      qx_PresetPermit : Bool := FALSE;   // Дозвіл виконання preset
      qx_PresetStart : Bool := FALSE;   // Одноцикловий імпульс запуску preset
      qd_PresetValueRaw : DInt := DINT#0;   // Значення preset, яке передається в блок енкодера
      qw_PresetStatus : Word := W#16#0000;   // Діагностичний код preset для діагностики/HMI
      qw_Status : Word := W#16#0000;   // Загальне діагностичне слово сіквенсера
      ql_TravelAfterReference_mm : LReal := 0.0;   // Шлях, пройдений після повторного проходження репера до повної зупинки, мм.
   END_VAR
   VAR
      stat_Step : UInt := UINT#0;   // Поточний внутрішній крок сіквенсера
      stat_PrevStep : UInt := UINT#0;   // Попередній крок для визначення зміни кроку
   END_VAR
   VAR RETAIN
      stat_Calibrated : Bool := FALSE;   // Запам'ятований результат успішної калібровки
   END_VAR
   VAR
      stat_MotionStarted : Bool := FALSE;   // Ознака, що під час процедури вже була команда руху
      stat_CompletedSteps : DWord := DWORD#0;   // Внутрішня бітова маска завершених кроків
      stat_StartOld : Bool := FALSE;   // Попередній стан команди Start
      stat_ResetOld : Bool := FALSE;   // Попередній стан команди Reset
      stat_AbortOld : Bool := FALSE;   // Попередній стан команди Abort
      stat_ReferenceOld : Bool := FALSE;   // Попередній стан сигналу 1K1
      tmr_TimeoutA : TON_TIME;   // Таймер очікування першої команди руху
      tmr_TimeoutB : TON_TIME;   // Таймер максимальної тривалості пошуку репера
      tmr_Standstill : TON_TIME;   // Таймер підтвердження повної зупинки ПЧ
      tmr_StepElapsed : TON_TIME;   // Таймер часу перебування на поточному кроці
      stat_RawAtReference : DInt := DINT#0;   // Raw-положення енкодера в момент повторного спадного фронту 1K1.
      stat_RawAtReferenceValid : Bool := FALSE;   // TRUE - raw-положення на репері успішно зафіксовано.
      stat_TravelAfterReference_mm : LReal := 0.0;   // Розрахований шлях від точки 1K1 до повної зупинки.
   END_VAR
   VAR_TEMP
      StartEdge : Bool;   // Передній фронт команди Start
      ResetEdge : Bool;   // Передній фронт команди Reset
      AbortEdge : Bool;   // Передній фронт команди Abort
      ReferenceFalling : Bool;   // Спадний фронт 1K1, TRUE → FALSE
      StepChanged : Bool;   // Поточний крок змінився
      StandstillCondition : Bool;   // ABS(DriveVelocity) <= StandstillSpeed
   END_VAR
BEGIN
   // ============================================================
   // 1. Формування фронтів
   // ============================================================

   #StartEdge :=
   #ix_Start
   AND NOT #stat_StartOld;

   #ResetEdge :=
   #ix_Reset
   AND NOT #stat_ResetOld;

   #AbortEdge :=
   #ix_Abort
   AND NOT #stat_AbortOld;

   // 1K1 заходить у PLC як нормально відкритий сигнал.
   // Проходження репера при підйомі: TRUE -> FALSE.
   #ReferenceFalling :=
   #stat_ReferenceOld
   AND NOT #ix_Reference1K1;


   // ============================================================
   // 2. Скидання
   // ============================================================

   IF #ResetEdge THEN

       #stat_Step := UINT#0;
       #stat_PrevStep := UINT#0;

       #stat_MotionStarted := FALSE;
       #stat_CompletedSteps := DWORD#0;

       // Clear data of the current reference procedure.
       #stat_RawAtReference := DINT#0;
       #stat_RawAtReferenceValid := FALSE;
       #stat_TravelAfterReference_mm := 0.0;

   END_IF;


   // ============================================================
   // 3. Timeout A
   // Очікування першої команди руху
   // ============================================================

   #tmr_TimeoutA(
                 IN :=
                 (#stat_Step = UINT#5)
                 OR (#stat_Step = UINT#20)
                 OR (#stat_Step = UINT#50)
                 OR (#stat_Step = UINT#70),
                 PT := #it_TimeoutA
   );


   // ============================================================
   // 4. Timeout B
   // Максимальний час пошуку реперної точки
   // ============================================================

   #tmr_TimeoutB(
                 IN :=
                 (#stat_Step = UINT#30)
                 OR (#stat_Step = UINT#80),
                 PT := #it_TimeoutB
   );


   // ============================================================
   // 5. Контроль повної зупинки ПЧ
   // ============================================================

   #StandstillCondition :=
   ABS(#ir_DriveVelocity_rpm)
   <= #ir_StandstillSpeed_rpm;

   #tmr_Standstill(
                   IN :=
                   (#stat_Step >= UINT#100)
                   AND (#stat_Step <= UINT#120)
                   AND #StandstillCondition,
                   PT := #it_StandstillConfirm
   );

   #qx_DriveStandstill :=
   #tmr_Standstill.Q;


   // ============================================================
   // 6. Таймер часу поточного кроку
   // ============================================================

   #StepChanged :=
   #stat_Step <> #stat_PrevStep;

   #tmr_StepElapsed(
                    IN :=
                    (#stat_Step > UINT#0)
                    AND (#stat_Step < UINT#130)
                    AND NOT #StepChanged,
                    PT := T#24d
   );

   #qt_StepElapsed :=
   #tmr_StepElapsed.ET;

   IF #StepChanged THEN
       #stat_PrevStep := #stat_Step;
   END_IF;


   // ============================================================
   // 7. Виходи за замовчуванням
   // ============================================================

   #qx_Active := FALSE;
   #qx_Aborted := FALSE;
   #qx_Fault := FALSE;

   #qx_BlockUp := TRUE;
   #qx_BlockDown := TRUE;
   #qx_QuickStop := FALSE;

   #qx_PresetServiceEnable := FALSE;
   #qx_PresetPermit := FALSE;
   #qx_PresetStart := FALSE;

   #qd_PresetValueRaw :=
   #id_PresetValueRaw;

   #qw_PresetStatus :=
   #iw_PresetStatus;


   // ============================================================
   // 8. Загальні умови аварійного завершення
   // ============================================================

   IF (#stat_Step > UINT#0)
       AND (#stat_Step < UINT#130)
   THEN

       // Ручне переривання процедури.
       IF #AbortEdge THEN

           #stat_Step := UINT#900;

           // Аварія ПЧ або активна аварія енкодера.
       ELSIF #ix_DriveFault
           OR #ix_EncoderFault
       THEN

           #stat_Step := UINT#910;

           // До запуску preset енкодер повинен бути готовим.
           // Після preset EncoderReady може короткочасно зникнути,
           // тому на кроках 110...120 ця умова тут не контролюється.
       ELSIF (#stat_Step < UINT#110)
           AND NOT #ix_EncoderReady
       THEN

           #stat_Step := UINT#910;

           // Не було команди руху за час Timeout A.
       ELSIF #tmr_TimeoutA.Q THEN

           #stat_Step := UINT#910;

           // Реперну процедуру не завершено за час Timeout B.
       ELSIF #tmr_TimeoutB.Q THEN

           #stat_Step := UINT#910;

       END_IF;

   END_IF;


   // ============================================================
   // 9. Основний сіквенсер
   // ============================================================

   CASE #stat_Step OF


           // --------------------------------------------------------
           // STEP 0
           // Калібровка неактивна
           // --------------------------------------------------------
       UINT#0:
           #qx_BlockUp := FALSE;
           #qx_BlockDown := FALSE;

           IF #StartEdge THEN

               #stat_Calibrated := FALSE;
               #stat_MotionStarted := FALSE;
               #stat_CompletedSteps := DWORD#0;
               #stat_RawAtReference := DINT#0;
               #stat_RawAtReferenceValid := FALSE;
               #stat_TravelAfterReference_mm := 0.0;

               // Якщо 1K1 знаходиться у нормальному стані,
               // починаємо стандартну процедуру калібровки.
               IF #ix_Reference1K1 THEN

                   #stat_Step := UINT#10;

                   // Якщо механізм знаходиться на / за точкою 1K1,
                   // спочатку необхідно відійти вниз від репера.
               ELSE

                   #stat_Step := UINT#5;

               END_IF;

           END_IF;

           // --------------------------------------------------------
           // STEP 5
           // Попередній відхід від 1K1
           //
           // Виконується тільки якщо процедура була запущена,
           // коли механізм знаходився на / за реперною точкою.
           // Після звільнення 1K1 починається стандартна
           // процедура калібровки з STEP 10.
           // --------------------------------------------------------
       UINT#5:

           #qx_Active := TRUE;

           // Рух вгору заборонений.
           // Дозволений тільки відхід вниз.
           #qx_BlockUp := TRUE;
           #qx_BlockDown := FALSE;

           // Фіксуємо факт початку руху.
           IF #ix_BtnDown THEN
               #stat_MotionStarted := TRUE;
           END_IF;

           // Після появи 1K1 механізм вже відійшов
           // від реперної точки.
           // Перед переходом оператор повинен
           // відпустити кнопку "Опускання".
           IF #ix_Reference1K1
               AND NOT #ix_BtnDown
           THEN

               // Починаємо стандартну процедуру.
               // Жодні біти CompletedSteps тут не встановлюються.
               #stat_Step := UINT#10;

           END_IF;

           // --------------------------------------------------------
           // STEP 10
           // Перевірка початкових умов
           // --------------------------------------------------------
       UINT#10:
           #qx_Active := TRUE;

           #qx_BlockUp := TRUE;
           #qx_BlockDown := TRUE;

           // Перед початком штатної процедури
           // обидві кнопки руху повинні бути відпущені.
           IF NOT #ix_BtnUp
               AND NOT #ix_BtnDown
           THEN

               #stat_CompletedSteps.%X0 := TRUE;

               #stat_Step := UINT#20;

           END_IF;

           // --------------------------------------------------------
           // STEP 20
           // Очікування першої команди підйому
           // --------------------------------------------------------
       UINT#20:

           #qx_Active := TRUE;

           #qx_BlockUp := FALSE;
           #qx_BlockDown := TRUE;

           IF #ix_BtnUp THEN

               #stat_MotionStarted := TRUE;
               #stat_CompletedSteps.%X1 := TRUE;

               #stat_Step := UINT#30;

           END_IF;


           // --------------------------------------------------------
           // STEP 30
           // Перший рух вгору до репера
           // --------------------------------------------------------
       UINT#30:

           #qx_Active := TRUE;

           #qx_BlockUp := FALSE;
           #qx_BlockDown := TRUE;

           IF #ReferenceFalling THEN

               #stat_CompletedSteps.%X2 := TRUE;

               #stat_Step := UINT#40;

           END_IF;


           // --------------------------------------------------------
           // STEP 40
           // Перше проходження 1K1
           // Очікування відпускання кнопки "Підйом"
           // --------------------------------------------------------
       UINT#40:

           #qx_Active := TRUE;

           #qx_BlockUp := TRUE;
           #qx_BlockDown := TRUE;

           IF NOT #ix_BtnUp THEN

               #stat_CompletedSteps.%X3 := TRUE;

               #stat_Step := UINT#50;

           END_IF;


           // --------------------------------------------------------
           // STEP 50
           // Відхід вниз від репера
           // --------------------------------------------------------
       UINT#50:

           #qx_Active := TRUE;

           #qx_BlockUp := TRUE;
           #qx_BlockDown := FALSE;

           IF #ix_BtnDown THEN
               #stat_MotionStarted := TRUE;
           END_IF;

           // Репер повинен бути звільнений,
           // а оператор повинен завершити відхід вниз.
           IF #ix_Reference1K1
               AND NOT #ix_BtnDown
           THEN

               #stat_CompletedSteps.%X4 := TRUE;

               #stat_Step := UINT#60;

           END_IF;


           // --------------------------------------------------------
           // STEP 60
           // Репер звільнений
           // Очікування відпускання кнопки "Опускання"
           // --------------------------------------------------------
       UINT#60:

           #qx_Active := TRUE;

           #qx_BlockUp := TRUE;
           #qx_BlockDown := TRUE;

           #stat_CompletedSteps.%X5 := TRUE;

           #stat_Step := UINT#70;


           // --------------------------------------------------------
           // STEP 70
           // Очікування повторної команди підйому
           // --------------------------------------------------------
       UINT#70:

           #qx_Active := TRUE;

           #qx_BlockUp := FALSE;
           #qx_BlockDown := TRUE;

           IF #ix_BtnUp THEN

               #stat_CompletedSteps.%X6 := TRUE;

               #stat_Step := UINT#80;

           END_IF;


           // --------------------------------------------------------
           // STEP 80
           // Повторний точний підхід до 1K1
           // --------------------------------------------------------
       UINT#80:

           #qx_Active := TRUE;

           #qx_BlockUp := FALSE;
           #qx_BlockDown := TRUE;

           IF #ReferenceFalling THEN

               // Save raw encoder position exactly at the
               // falling edge of reference switch 1K1.
               IF #ix_PositionScaleValid THEN

                   #stat_RawAtReference := #id_ActualPositionRaw;
                   #stat_RawAtReferenceValid := TRUE;

                   #stat_CompletedSteps.%X7 := TRUE;

                   #stat_Step := UINT#90;

               ELSE

                   // Position scaling is not valid.
                   #stat_RawAtReferenceValid := FALSE;
                   #stat_Step := UINT#910;

               END_IF;

           END_IF;

           // --------------------------------------------------------
           // STEP 90
           // Формування Quick Stop
           // --------------------------------------------------------
       UINT#90:

           #qx_Active := TRUE;

           #qx_BlockUp := TRUE;
           #qx_BlockDown := TRUE;
           #qx_QuickStop := TRUE;

           #stat_CompletedSteps.%X8 := TRUE;

           // Крок утримується один цикл PLC.
           #stat_Step := UINT#100;


           // --------------------------------------------------------
           // STEP 100
           // Очікування повної зупинки ПЧ
           // --------------------------------------------------------
       UINT#100:

           #qx_Active := TRUE;

           #qx_BlockUp := TRUE;
           #qx_BlockDown := TRUE;

           // OFF3 утримується до підтвердженої зупинки.
           #qx_QuickStop := TRUE;

           IF #qx_DriveStandstill
               AND NOT #ix_BtnUp
               AND NOT #ix_BtnDown
           THEN

               // Reference position must be saved before calculation.
               IF #stat_RawAtReferenceValid
                   AND #ix_PositionScaleValid
               THEN

                   // Calculate travel from the reference switch
                   // to the final standstill position.
                   #stat_TravelAfterReference_mm :=
                   (
                   DINT_TO_LREAL(#id_ActualPositionRaw)
                   - DINT_TO_LREAL(#stat_RawAtReference)
                   )
                   * #il_Scale_mm_per_count;

                   #stat_CompletedSteps.%X9 := TRUE;

                   #stat_Step := UINT#110;

               ELSE

                   // Reference data or scaling is not valid.
                   #stat_Step := UINT#910;

               END_IF;

           END_IF;


           // --------------------------------------------------------
           // STEP 110
           // Запуск preset
           // --------------------------------------------------------
       UINT#110:

           #qx_Active := TRUE;

           #qx_BlockUp := TRUE;
           #qx_BlockDown := TRUE;

           #qx_PresetServiceEnable := TRUE;

           #qx_PresetPermit :=
           #qx_DriveStandstill
           AND NOT #ix_BtnUp
           AND NOT #ix_BtnDown
           AND #ix_EncoderReady
           AND NOT #ix_EncoderFault
           AND NOT #ix_DriveFault;

           // PresetStart активний тільки один цикл.
           IF #qx_PresetPermit THEN

               #qx_PresetStart := TRUE;

               #stat_CompletedSteps.%X10 := TRUE;

               #stat_Step := UINT#120;

           END_IF;


           // --------------------------------------------------------
           // STEP 120
           // Очікування завершення preset
           // --------------------------------------------------------
       UINT#120:

           #qx_Active := TRUE;

           #qx_BlockUp := TRUE;
           #qx_BlockDown := TRUE;

           #qx_PresetServiceEnable := TRUE;

           // Після запуску preset EncoderReady може короткочасно
           // стати FALSE через invalid position/velocity.
           // Тому тут не використовуємо EncoderReady
           // як умову помилки процедури.

           #qx_PresetPermit :=
           #qx_DriveStandstill
           AND NOT #ix_BtnUp
           AND NOT #ix_BtnDown
           AND NOT #ix_EncoderFault
           AND NOT #ix_DriveFault;

           IF #ix_PresetDone THEN

               #stat_CompletedSteps.%X11 := TRUE;

               #stat_Step := UINT#130;

           ELSIF #ix_PresetError THEN

               #stat_Step := UINT#910;

           END_IF;


           // --------------------------------------------------------
           // STEP 130
           // Калібровка успішно завершена
           // --------------------------------------------------------
       UINT#130:

           #qx_BlockUp := FALSE;
           #qx_BlockDown := FALSE;

           #stat_Calibrated := TRUE;
           #stat_CompletedSteps.%X12 := TRUE;

           // Успішний статус калібровки зберігається.
           // Він скидається тільки при запуску нової повної калібровки.

           // --------------------------------------------------------
           // STEP 900
           // Ручне переривання
           // --------------------------------------------------------
       UINT#900:

           #qx_Aborted := TRUE;

           #qx_BlockUp := TRUE;
           #qx_BlockDown := TRUE;

           #qx_QuickStop := TRUE;


           // --------------------------------------------------------
           // STEP 910
           // Помилка процедури
           // --------------------------------------------------------
       UINT#910:

           #qx_Fault := TRUE;

           #qx_BlockUp := TRUE;
           #qx_BlockDown := TRUE;

           #qx_QuickStop := TRUE;


           // --------------------------------------------------------
           // Некоректний номер кроку
           // --------------------------------------------------------
       ELSE

           #stat_Step := UINT#910;

   END_CASE;


   // ============================================================
   // 10. Основні статуси
   // ============================================================

   #qu_CurrentStep :=
   #stat_Step;

   #qd_CompletedSteps :=
   #stat_CompletedSteps;

   // Нормальна та форсована калібровка формують один вихід.
   #qx_Calibrated :=
   #stat_Calibrated
   OR #ix_ForceCalibrated;

   #ql_TravelAfterReference_mm :=
   #stat_TravelAfterReference_mm;

   // ============================================================
   // 11. Активний таймер для HMI
   // ============================================================

   #qt_ActiveTimerElapsed := T#0ms;
   #qt_ActiveTimerPreset := T#0ms;
   #qt_ActiveTimerRemaining := T#0ms;


   // Timeout A.
   IF (#stat_Step = UINT#5)
       OR (#stat_Step = UINT#20)
       OR (#stat_Step = UINT#50)
       OR (#stat_Step = UINT#70)
   THEN

       #qt_ActiveTimerElapsed :=
       #tmr_TimeoutA.ET;

       #qt_ActiveTimerPreset :=
       #it_TimeoutA;

       IF #tmr_TimeoutA.ET < #it_TimeoutA THEN

           #qt_ActiveTimerRemaining :=
           #it_TimeoutA - #tmr_TimeoutA.ET;

       END_IF;


       // Timeout B.
   ELSIF 
       (#stat_Step = UINT#30)
       OR (#stat_Step = UINT#80)
   THEN

       #qt_ActiveTimerElapsed :=
       #tmr_TimeoutB.ET;

       #qt_ActiveTimerPreset :=
       #it_TimeoutB;

       IF #tmr_TimeoutB.ET < #it_TimeoutB THEN

           #qt_ActiveTimerRemaining :=
           #it_TimeoutB - #tmr_TimeoutB.ET;

       END_IF;


       // Standstill.
   ELSIF #stat_Step = UINT#100 THEN

       #qt_ActiveTimerElapsed :=
       #tmr_Standstill.ET;

       #qt_ActiveTimerPreset :=
       #it_StandstillConfirm;

       IF #tmr_Standstill.ET < #it_StandstillConfirm THEN

           #qt_ActiveTimerRemaining :=
           #it_StandstillConfirm - #tmr_Standstill.ET;

       END_IF;

   END_IF;


   // ============================================================
   // 12. Діагностичне слово
   //
   // Bit 0  - процедура активна
   // Bit 1  - механізм калібрований
   // Bit 2  - процедура перервана
   // Bit 3  - помилка процедури
   // Bit 4  - Drive Standstill
   // Bit 5  - Preset Busy
   // Bit 6  - Preset Error
   // Bit 8  - Timeout A
   // Bit 9  - Timeout B
   // Bit 10 - Drive Fault
   // Bit 11 - Encoder Fault
   // Bit 12 - Encoder Not Ready
   // ============================================================

   #qw_Status := W#16#0000;

   IF #qx_Active THEN
       #qw_Status := #qw_Status OR W#16#0001;
   END_IF;

   IF #qx_Calibrated THEN
       #qw_Status := #qw_Status OR W#16#0002;
   END_IF;

   IF #qx_Aborted THEN
       #qw_Status := #qw_Status OR W#16#0004;
   END_IF;

   IF #qx_Fault THEN
       #qw_Status := #qw_Status OR W#16#0008;
   END_IF;

   IF #qx_DriveStandstill THEN
       #qw_Status := #qw_Status OR W#16#0010;
   END_IF;

   IF #ix_PresetBusy THEN
       #qw_Status := #qw_Status OR W#16#0020;
   END_IF;

   IF #ix_PresetError THEN
       #qw_Status := #qw_Status OR W#16#0040;
   END_IF;

   IF #tmr_TimeoutA.Q THEN
       #qw_Status := #qw_Status OR W#16#0100;
   END_IF;

   IF #tmr_TimeoutB.Q THEN
       #qw_Status := #qw_Status OR W#16#0200;
   END_IF;

   IF #ix_DriveFault THEN
       #qw_Status := #qw_Status OR W#16#0400;
   END_IF;

   IF #ix_EncoderFault THEN
       #qw_Status := #qw_Status OR W#16#0800;
   END_IF;

   IF NOT #ix_EncoderReady THEN
       #qw_Status := #qw_Status OR W#16#1000;
   END_IF;


   // ============================================================
   // 13. Запам'ятовування станів
   // ============================================================

   #stat_StartOld :=
   #ix_Start;

   #stat_ResetOld :=
   #ix_Reset;

   #stat_AbortOld :=
   #ix_Abort;

   #stat_ReferenceOld :=
   #ix_Reference1K1;
END_FUNCTION_BLOCK

FUNCTION_BLOCK "FB_HoistCalibrationDiag"   // FB711, SCL
{ S7_Optimized_Access := 'TRUE' }
VERSION : 0.1
   VAR_INPUT
      ix_Reset : Bool := FALSE;   // Скидання зафіксованих діагностичних помилок
      ix_EncoderReady : Bool := FALSE;   // Енкодер 1BR готовий
      ix_EncoderFault : Bool := FALSE;   // Помилка енкодера
      ix_CommunicationFault : Bool := FALSE;   // Помилка зв'язку з енкодером
      il_Position_mm : LReal := 0.0;   // Поточна координата механізму, мм
      ix_MoveCommand : Bool := FALSE;   // Дійсна команда руху механізму
      ix_DriveFault : Bool := FALSE;   // Аварія привода
      ir_DriveVelocity_rpm : Real := 0.0;   // Фактична швидкість привода
      ix_CalibrationActive : Bool := FALSE;   // Процедура калібровки активна
      ix_Calibrated : Bool := FALSE;   // Механізм відкалібровано
      ix_ManualDriveActive : Bool := FALSE;   // Ручний привод/розгальмування активний; поки подаємо FALSE
      il_NoMoveThreshold_mm : LReal := 5.0;   // Допустима зміна положення без команди руху
      il_MoveMinDelta_mm : LReal := 1.0;   // Мінімальна зміна положення для підтвердження роботи енкодера
      it_MoveUpdateTimeout : Time := T#1s;   // Максимальний час без зміни положення при команді руху
      ir_StandstillSpeed_rpm : Real := 5.0;   // Поріг повної зупинки
      it_StandstillConfirm : Time := T#500ms;   // Час підтвердження повної зупинки
      il_StartupTolerance_mm : LReal := 5.0;   // Допуск порівняння положення після запуску PLC
   END_VAR
   VAR_OUTPUT
      qx_EncoderControlHealthy : Bool := FALSE;   // Енкодер і зв'язок справні
      qx_StartupDataConsistent : Bool := TRUE;   // Положення після старту PLC узгоджене
      qx_NoMovementWithoutCommand : Bool := TRUE;   // Не виявлено переміщення без команди
      qx_NoManualMovementDetected : Bool := TRUE;   // Не виявлено нештатного руху без ручного приводу
      qx_EncoderUpdatesDuringMotion : Bool := TRUE;   // Енкодер змінює значення при команді руху
      qx_EncoderReplacementNotDetected : Bool := TRUE;   // Зарезервовано; поки завжди норма
      qx_DiagnosticsHealthy : Bool := FALSE;   // Усі реально реалізовані контролі в нормі
      qx_DriveStandstill : Bool := FALSE;   // Підтверджена повна зупинка
      ql_PositionDeltaStopped_mm : LReal := 0.0;   // Зміна позиції від точки останньої зупинки
      ql_PositionDeltaMotion_mm : LReal := 0.0;   // Зміна позиції для watchdog руху
   END_VAR
   VAR RETAIN
      stat_SavedPosition_mm : LReal := 0.0;   // Положення, збережене до перезапуску
      stat_SavedPositionValid : Bool := FALSE;   // Ознака валідності збереженого положення
   END_VAR
   VAR
      stat_StartupChecked : Bool := FALSE;   // Перевірка після запуску PLC виконана
      stat_StopReference_mm : LReal := 0.0;   // Базова позиція після зупинки
      stat_StopReferenceValid : Bool := FALSE;   // Базова позиція зупинки валідна
      stat_MoveReference_mm : LReal := 0.0;   // Базова позиція для watchdog руху
      stat_MoveMonitorActive : Bool := FALSE;   // Контроль зміни позиції при русі активний
      stat_WasMoving : Bool := FALSE;   // Ознака, що механізм до цього рухався
      stat_StartupMismatchFault : Bool := FALSE;   // Виявлена невідповідність положення після запуску
      stat_MoveWithoutCommandFault : Bool := FALSE;   // Виявлено зміну положення без команди руху
      stat_NoUpdateDuringMotionFault : Bool := FALSE;   // Не виявлено зміни положення при команді руху
      stat_CalibratedOld : Bool := FALSE;   // Попередній стан сигналу Calibrated
      tmr_Standstill : TON_TIME;   // Таймер підтвердження повної зупинки
      tmr_MoveUpdate : TON_TIME;   // Watchdog оновлення положення при русі
   END_VAR
   VAR_TEMP
      EncoderHealthy : Bool;   // Поточна ознака справності енкодера та зв’язку
      StandstillCondition : Bool;   // Умова низької швидкості для визначення повної зупинки
      CalibratedRising : Bool;   // Передній фронт статусу Calibrated
      MoveDeltaReached : Bool;   // Положення змінилося не менше заданого мінімуму
      MoveWatchdogEnable : Bool;   // Дозвіл роботи watchdog контролю зміни положення
   END_VAR
BEGIN
   // ============================================================
   // 1. Загальна справність енкодера
   // ============================================================

   #EncoderHealthy :=
   #ix_EncoderReady
   AND NOT #ix_EncoderFault
   AND NOT #ix_CommunicationFault;

   #qx_EncoderControlHealthy :=
   #EncoderHealthy;


   // ============================================================
   // 2. Визначення повної зупинки
   // ============================================================

   #StandstillCondition :=
   ABS(#ir_DriveVelocity_rpm)
   <= #ir_StandstillSpeed_rpm;

   #tmr_Standstill(
                   IN :=
                   #StandstillCondition
                   AND NOT #ix_MoveCommand,
                   PT := #it_StandstillConfirm
   );

   #qx_DriveStandstill :=
   #tmr_Standstill.Q;


   // ============================================================
   // 3. Фронт отримання статусу "Калібровано"
   // ============================================================

   #CalibratedRising :=
   #ix_Calibrated
   AND NOT #stat_CalibratedOld;


   // ============================================================
   // 4. Reset діагностики
   // ============================================================

   IF #ix_Reset THEN

       #stat_StartupMismatchFault := FALSE;
       #stat_MoveWithoutCommandFault := FALSE;
       #stat_NoUpdateDuringMotionFault := FALSE;

       #stat_StopReferenceValid := FALSE;
       #stat_MoveMonitorActive := FALSE;

   END_IF;


   // ============================================================
   // 5. Перевірка положення після запуску PLC
   //
   // Виконується один раз після появи валідних даних енкодера.
   // Retain-позиція ще не перезаписується до завершення перевірки.
   // ============================================================

   IF NOT #stat_StartupChecked
       AND #EncoderHealthy
   THEN

       IF #stat_SavedPositionValid THEN

           IF ABS(#il_Position_mm - #stat_SavedPosition_mm)
               > #il_StartupTolerance_mm
           THEN

               #stat_StartupMismatchFault := TRUE;

           END_IF;

       ELSE

           // Перший запуск: попереднього значення ще немає.
           #stat_SavedPosition_mm :=
           #il_Position_mm;

           #stat_SavedPositionValid := TRUE;

       END_IF;

       #stat_StartupChecked := TRUE;

       // Початкова база для контролю нерухомості.
       #stat_StopReference_mm :=
       #il_Position_mm;

       #stat_StopReferenceValid := TRUE;

   END_IF;


   // ============================================================
   // 6. Після успішної калібровки
   //
   // Preset штатно змінює координату без фізичного руху.
   // Тому після калібровки формуємо нову базову позицію.
   // ============================================================

   IF #CalibratedRising
       AND #EncoderHealthy
   THEN

       #stat_StopReference_mm :=
       #il_Position_mm;

       #stat_StopReferenceValid := TRUE;

       #stat_SavedPosition_mm :=
       #il_Position_mm;

       #stat_SavedPositionValid := TRUE;

       // Калібровка формує нову достовірну координату.
       #stat_StartupMismatchFault := FALSE;
       #stat_MoveWithoutCommandFault := FALSE;
       #stat_NoUpdateDuringMotionFault := FALSE;

   END_IF;


   // ============================================================
   // 7. Запам'ятовування факту руху
   // ============================================================

   IF #ix_MoveCommand THEN
       #stat_WasMoving := TRUE;
   END_IF;


   // ============================================================
   // 8. Формування нової бази після завершення руху
   //
   // Після підтвердженої повної зупинки зберігаємо положення.
   // ============================================================

   IF #qx_DriveStandstill
       AND #stat_WasMoving
       AND #EncoderHealthy
       AND NOT #ix_CalibrationActive
   THEN

       #stat_StopReference_mm :=
       #il_Position_mm;

       #stat_StopReferenceValid := TRUE;

       #stat_SavedPosition_mm :=
       #il_Position_mm;

       #stat_SavedPositionValid := TRUE;

       #stat_WasMoving := FALSE;

   END_IF;


   // ============================================================
   // 9. Контроль зміни положення без команди руху
   //
   // Контроль виконується тільки:
   // - після підтвердженої повної зупинки;
   // - без команди руху;
   // - без ручного приводу;
   // - поза процедурою калібровки.
   // ============================================================

   #ql_PositionDeltaStopped_mm := 0.0;

   IF #qx_DriveStandstill
       AND NOT #ix_MoveCommand
       AND NOT #ix_ManualDriveActive
       AND NOT #ix_CalibrationActive
       AND #EncoderHealthy
       AND #stat_StopReferenceValid
   THEN

       #ql_PositionDeltaStopped_mm :=
       ABS(#il_Position_mm - #stat_StopReference_mm);

       IF #ql_PositionDeltaStopped_mm
           > #il_NoMoveThreshold_mm
       THEN

           #stat_MoveWithoutCommandFault := TRUE;

       END_IF;

   END_IF;


   // ============================================================
   // 10. Контроль оновлення енкодера під час руху
   //
   // Якщо є дійсна команда руху і немає аварії привода,
   // координата повинна змінюватись не менш ніж на задану величину
   // протягом MoveUpdateTimeout.
   // ============================================================

   IF #ix_MoveCommand
       AND NOT #ix_DriveFault
       AND #EncoderHealthy
   THEN

       IF NOT #stat_MoveMonitorActive THEN

           #stat_MoveReference_mm :=
           #il_Position_mm;

           #stat_MoveMonitorActive := TRUE;

       END_IF;

       #ql_PositionDeltaMotion_mm :=
       ABS(#il_Position_mm - #stat_MoveReference_mm);

       #MoveDeltaReached :=
       #ql_PositionDeltaMotion_mm >= #il_MoveMinDelta_mm;

       IF #MoveDeltaReached THEN

           // Є нормальна зміна координати.
           // Починаємо наступний інтервал контролю.
           #stat_MoveReference_mm :=
           #il_Position_mm;

       END_IF;

   ELSE

       #stat_MoveMonitorActive := FALSE;
       #ql_PositionDeltaMotion_mm := 0.0;
       #MoveDeltaReached := FALSE;

   END_IF;


   // Watchdog працює, поки координата не змінилася
   // на необхідну величину.
   #MoveWatchdogEnable :=
   #stat_MoveMonitorActive
   AND NOT #MoveDeltaReached;

   #tmr_MoveUpdate(
                   IN := #MoveWatchdogEnable,
                   PT := #it_MoveUpdateTimeout
   );

   IF #tmr_MoveUpdate.Q THEN
       #stat_NoUpdateDuringMotionFault := TRUE;
   END_IF;


   // ============================================================
   // 11. Позитивні діагностичні виходи
   // ============================================================

   #qx_StartupDataConsistent :=
   NOT #stat_StartupMismatchFault;

   #qx_NoMovementWithoutCommand :=
   NOT #stat_MoveWithoutCommandFault;

   // Поки окремого сигналу ручного приводу немає.
   // Контроль використовує його як дозвільну умову.
   #qx_NoManualMovementDetected :=
   NOT #stat_MoveWithoutCommandFault;

   #qx_EncoderUpdatesDuringMotion :=
   NOT #stat_NoUpdateDuringMotionFault;


   // ============================================================
   // 12. Контроль фізичної заміни енкодера
   //
   // Поки не реалізований.
   // До появи надійного способу ідентифікації енкодера
   // сигнал примусово встановлений у стан "Норма".
   // ============================================================

   #qx_EncoderReplacementNotDetected := TRUE;


   // ============================================================
   // 13. Загальний результат
   //
   // Зарезервований контроль фізичної заміни енкодера
   // поки не бере участі у DiagnosticsHealthy.
   // ============================================================

   #qx_DiagnosticsHealthy :=
   #qx_EncoderControlHealthy
   AND #qx_StartupDataConsistent
   AND #qx_NoMovementWithoutCommand
   AND #qx_NoManualMovementDetected
   AND #qx_EncoderUpdatesDuringMotion;


   // ============================================================
   // 14. Запам'ятовування станів
   // ============================================================

   #stat_CalibratedOld :=
   #ix_Calibrated;
END_FUNCTION_BLOCK

// folder: 700_Calibration/Trolley

FUNCTION_BLOCK "FB_TrolleyCalibration"   // FB702, SCL
{ S7_Optimized_Access := 'TRUE' }
VERSION : 0.1
   VAR_INPUT
      ix_Start : Bool := FALSE;   // Запуск процедури калібровки
      ix_Reset : Bool := FALSE;   // Скидання сіквенсера поточної процедури калібровки (без зміни статусу)
      ix_Abort : Bool := FALSE;   // Ручне переривання процедури
      ix_ForceCalibrated : Bool := FALSE;   // Примусове встановлення статусу калібровки для ПНР
      ix_HoistCalibrated : Bool := FALSE;   // Підйом відкалібрований
      il_HoistPosition_mm : LReal := 0.0;   // Поточна координата підйому
      il_HoistPositionMin_mm : LReal := 23750.0;   // Нижня межа допустимої позиції підйому
      il_HoistPositionMax_mm : LReal := 23900.0;   // Верхня межа допустимої позиції підйому
      ix_Reference3K1 : Bool := FALSE;   // Реперний сигнал 3K1
      ix_BtnForward : Bool := FALSE;   // Команда «Вперед»
      ix_BtnBackward : Bool := FALSE;   // Команда «Назад»
      ix_DriveFault : Bool := FALSE;   // Аварія ПЧ візка
      ir_DriveVelocity_rpm : Real := 0.0;   // Фактична швидкість ПЧ
      ix_EncoderReady : Bool := FALSE;   // Енкодер 3BR готовий
      ix_EncoderFault : Bool := FALSE;   // Помилка енкодера 3BR
      ix_PresetBusy : Bool := FALSE;   // Preset активний
      ix_PresetDone : Bool := FALSE;   // Preset успішно завершено
      ix_PresetError : Bool := FALSE;   // Помилка preset
      iw_PresetStatus : Word := W#16#0000;   // Статус preset
      id_PresetValueRaw : DInt := DINT#119305476;   // Розраховане raw-значення для preset енкодера 3BR.
      it_TimeoutA : Time := T#1m;   // Час очікування першої команди
      it_TimeoutB : Time := T#5m;   // Максимальний час реперної процедури
      ir_StandstillSpeed_rpm : Real := 5.0;   // Поріг standstill
      it_StandstillConfirm : Time := T#500ms;   // Підтвердження standstill
      id_ActualPositionRaw : DInt := DINT#0;   // Поточне абсолютне raw-положення енкодера 3BR.
      il_Scale_mm_per_count : LReal := 0.0;   // Коефіцієнт перетворення raw-count у мм для енкодера 3BR.
      ix_PositionScaleValid : Bool := FALSE;   // TRUE — масштабування положення енкодера 3BR налаштоване коректно.
   END_VAR
   VAR_OUTPUT
      qx_Active : Bool := FALSE;   // Процедура активна
      qx_Calibrated : Bool := FALSE;   // Візок калібрований
      qx_Aborted : Bool := FALSE;   // Процедуру перервано
      qx_Fault : Bool := FALSE;   // Помилка процедури
      qx_PrerequisitesNotOK : Bool := FALSE;   // Не виконані попередні умови для калібровки візка
      qu_CurrentStep : UInt := UINT#0;   // Поточний крок
      qd_CompletedSteps : DWord := DWORD#0;   // Завершені кроки
      qt_StepElapsed : Time := T#0ms;   // Час поточного кроку
      qt_ActiveTimerElapsed : Time := T#0ms;   // Час активного таймера
      qt_ActiveTimerPreset : Time := T#0ms;   // Уставка таймера
      qt_ActiveTimerRemaining : Time := T#0ms;   // Залишок часу
      qx_BlockForward : Bool := FALSE;   // Заборона руху вперед
      qx_BlockBackward : Bool := FALSE;   // Заборона руху назад
      qx_QuickStop : Bool := FALSE;   // Запит Quick Stop
      qx_DriveStandstill : Bool := FALSE;   // Підтверджена зупинка
      qx_PresetServiceEnable : Bool := FALSE;   // Дозвіл сервісного preset
      qx_PresetPermit : Bool := FALSE;   // Умови preset виконані
      qx_PresetStart : Bool := FALSE;   // Одноцикловий запуск preset
      qd_PresetValueRaw : DInt := DINT#0;   // Значення preset
      qw_PresetStatus : Word := W#16#0000;   // Статус preset
      qw_Status : Word := W#16#0000;   // Загальний статус
      ql_TravelAfterReference_mm : LReal := 0.0;   // Шлях, пройдений після повторного проходження 3K1 до повної зупинки, мм.
   END_VAR
   VAR
      stat_Step : UInt := UINT#0;   // Поточний внутрішній крок сіквенсера
      stat_PrevStep : UInt := UINT#0;   // Попередній крок для визначення зміни кроку
   END_VAR
   VAR RETAIN
      stat_Calibrated : Bool := FALSE;   // Запам'ятований результат успішної калібровки
   END_VAR
   VAR
      stat_MotionStarted : Bool := FALSE;   // Ознака, що під час процедури вже була команда руху
      stat_CompletedSteps : DWord := DWORD#0;   // Внутрішня бітова маска завершених кроків
      stat_StartOld : Bool := FALSE;   // Попередній стан команди Start
      stat_ResetOld : Bool := FALSE;   // Попередній стан команди Reset
      stat_AbortOld : Bool := FALSE;   // Попередній стан команди Abort
      stat_ReferenceOld : Bool := FALSE;   // Попередній стан сигналу 1K1
      tmr_TimeoutA : TON_TIME;   // Таймер очікування першої команди руху
      tmr_TimeoutB : TON_TIME;   // Таймер максимальної тривалості пошуку репера
      tmr_Standstill : TON_TIME;   // Таймер підтвердження повної зупинки ПЧ
      tmr_StepElapsed : TON_TIME;   // Таймер часу перебування на поточному кроці
      stat_RawAtReference : DInt := DINT#0;   // Raw-положення енкодера в момент повторного спадного фронту 3K1.
      stat_RawAtReferenceValid : Bool := FALSE;   // TRUE - raw-положення в точці 3K1 успішно зафіксовано.
      stat_TravelAfterReference_mm : LReal := 0.0;   // Розрахований шлях від 3K1 до повної зупинки.
   END_VAR
   VAR_TEMP
      StartEdge : Bool;
      ResetEdge : Bool;
      AbortEdge : Bool;
      ReferenceFalling : Bool;
      StepChanged : Bool;
      StandstillCondition : Bool;
      HoistPositionOK : Bool;
   END_VAR
BEGIN
   // ============================================================
   // 1. Формування фронтів
   // ============================================================

   #StartEdge :=
   #ix_Start
   AND NOT #stat_StartOld;

   #ResetEdge :=
   #ix_Reset
   AND NOT #stat_ResetOld;

   #AbortEdge :=
   #ix_Abort
   AND NOT #stat_AbortOld;

   // 3K1: проходження репера при русі вперед TRUE -> FALSE
   #ReferenceFalling :=
   #stat_ReferenceOld
   AND NOT #ix_Reference3K1;


   // ============================================================
   // 2. Перевірка положення підйому
   // ============================================================

   #HoistPositionOK :=
   #ix_HoistCalibrated
   AND (#il_HoistPosition_mm >= #il_HoistPositionMin_mm)
   AND (#il_HoistPosition_mm <= #il_HoistPositionMax_mm);

   #qx_PrerequisitesNotOK := NOT #HoistPositionOK;

   // ============================================================
   // 3. Reset
   // ============================================================

   IF #ResetEdge THEN

       #stat_Step := UINT#0;
       #stat_PrevStep := UINT#0;

       #stat_MotionStarted := FALSE;
       #stat_CompletedSteps := DWORD#0;

       // Очищення даних поточної реперної процедури.
       #stat_RawAtReference := DINT#0;
       #stat_RawAtReferenceValid := FALSE;
       #stat_TravelAfterReference_mm := 0.0;

   END_IF;


   // ============================================================
   // 4. Timeout A
   // ============================================================

   #tmr_TimeoutA(
                 IN :=
                 (#stat_Step = UINT#5)
                 OR (#stat_Step = UINT#20)
                 OR (#stat_Step = UINT#50)
                 OR (#stat_Step = UINT#70),
                 PT := #it_TimeoutA
   );


   // ============================================================
   // 5. Timeout B
   // ============================================================

   #tmr_TimeoutB(
                 IN :=
                 (#stat_Step = UINT#30)
                 OR (#stat_Step = UINT#80),
                 PT := #it_TimeoutB
   );


   // ============================================================
   // 6. Контроль повної зупинки ПЧ
   // ============================================================

   #StandstillCondition :=
   ABS(#ir_DriveVelocity_rpm)
   <= #ir_StandstillSpeed_rpm;

   #tmr_Standstill(
                   IN :=
                   (#stat_Step >= UINT#100)
                   AND (#stat_Step <= UINT#120)
                   AND #StandstillCondition,
                   PT := #it_StandstillConfirm
   );

   #qx_DriveStandstill :=
   #tmr_Standstill.Q;


   // ============================================================
   // 7. Таймер поточного кроку
   // ============================================================

   #StepChanged :=
   #stat_Step <> #stat_PrevStep;

   #tmr_StepElapsed(
                    IN :=
                    (#stat_Step > UINT#0)
                    AND (#stat_Step < UINT#130)
                    AND NOT #StepChanged,
                    PT := T#24d
   );

   #qt_StepElapsed :=
   #tmr_StepElapsed.ET;

   IF #StepChanged THEN
       #stat_PrevStep := #stat_Step;
   END_IF;


   // ============================================================
   // 8. Виходи за замовчуванням
   // ============================================================

   #qx_Active := FALSE;
   #qx_Aborted := FALSE;
   #qx_Fault := FALSE;

   #qx_BlockForward := TRUE;
   #qx_BlockBackward := TRUE;

   #qx_QuickStop := FALSE;

   #qx_PresetServiceEnable := FALSE;
   #qx_PresetPermit := FALSE;
   #qx_PresetStart := FALSE;

   #qd_PresetValueRaw :=
   #id_PresetValueRaw;

   #qw_PresetStatus :=
   #iw_PresetStatus;


   // ============================================================
   // 9. Загальні умови аварійного завершення
   // ============================================================

   IF (#stat_Step > UINT#0)
       AND (#stat_Step < UINT#130)
   THEN

       IF #AbortEdge THEN

           #stat_Step := UINT#900;

       ELSIF #ix_DriveFault
           OR #ix_EncoderFault
       THEN

           #stat_Step := UINT#910;

           // Підйом повинен залишатися каліброваним
           // та знаходитися в допустимій зоні.
       ELSIF NOT #HoistPositionOK THEN

           #stat_Step := UINT#910;

           // До запуску preset енкодер повинен бути готовим.
       ELSIF (#stat_Step < UINT#110)
           AND NOT #ix_EncoderReady
       THEN

           #stat_Step := UINT#910;

       ELSIF #tmr_TimeoutA.Q THEN

           #stat_Step := UINT#910;

       ELSIF #tmr_TimeoutB.Q THEN

           #stat_Step := UINT#910;

       END_IF;

   END_IF;


   // ============================================================
   // 10. Основний сіквенсер
   // ============================================================

   CASE #stat_Step OF


